LIN {X 0,Y 193.317,Z 565.534,A -85,B 0,C 180,E1 11170.664,E2 11170.664} C_VEL
LIN {X 0,Y 192.779,Z 572.927,A -85,B 0,C 180,E1 11165.955,E2 11165.955} C_VEL
LIN {X 0,Y 192.758,Z 579.081,A -85,B 0,C 180,E1 11160.892,E2 11160.892} C_VEL
LIN {X 0,Y 193.304,Z 583.795,A -85,B 0,C 180,E1 11155.551,E2 11155.551} C_VEL
LIN {X 0,Y 194.84,Z 586.974,A -85,B 0,C 180,E1 11149.952,E2 11149.952} C_VEL
LIN {X 0,Y 197.91,Z 588.494,A -85,B 0,C 180,E1 11144.169,E2 11144.169} C_VEL
LIN {X 0,Y 202.718,Z 588.212,A -85,B 0,C 180,E1 11138.594,E2 11138.594} C_VEL
LIN {X 0,Y 209.71,Z 586.058,A -85,B 0,C 180,E1 11133.068,E2 11133.068} C_VEL
LIN {X 0,Y 218.66,Z 582.103,A -85,B 0,C 180,E1 11127.966,E2 11127.966} C_VEL
LIN {X 0,Y 230.621,Z 575.806,A -85,B 0,C 180,E1 11122.942,E2 11122.942} C_VEL
LIN {X 0,Y 243.425,Z 568.326,A -85,B 0,C 180,E1 11118.835,E2 11118.835} C_VEL
LIN {X 0,Y 227.864,Z 579.481,A -85,B 0,C 180,E1 11114.244,E2 11114.244} C_VEL
LIN {X 0,Y 214.538,Z 589.641,A -85,B 0,C 180,E1 11108.648,E2 11108.648} C_VEL
LIN {X 0,Y 203.983,Z 598.452,A -85,B 0,C 180,E1 11101.966,E2 11101.966} C_VEL
LIN {X 0,Y 197.328,Z 604.793,A -85,B 0,C 180,E1 11095.192,E2 11095.192} C_VEL
LIN {X 0,Y 193.795,Z 608.88,A -85,B 0,C 180,E1 11088.658,E2 11088.658} C_VEL
LIN {X 0,Y 192.5,Z 611.05,A -85,B 0,C 180,E1 11082.298,E2 11082.298} C_VEL
LIN {X 0,Y 192.502,Z 613.904,A -85,B 0,C 180,E1 11076.264,E2 11076.264} C_VEL
LIN {X 0,Y 192.758,Z 614.861,A -85,B 0,C 180,E1 11071.488,E2 11071.488} C_VEL
LIN {X 0,Y 192.704,Z 614.748,A -85,B 0,C 180,E1 11067.325,E2 11067.325} C_VEL
LIN {X 0,Y 192.429,Z 613.273,A -85,B 0,C 180,E1 11062.238,E2 11062.238} C_VEL
LIN {X 0,Y 192.571,Z 610.294,A -85,B 0,C 180,E1 11056.796,E2 11056.796} C_VEL
LIN {X 0,Y 193.943,Z 605.17,A -85,B 0,C 180,E1 11050.737,E2 11050.737} C_VEL
LIN {X 0,Y 196.931,Z 598.058,A -85,B 0,C 180,E1 11044.757,E2 11044.757} C_VEL
LIN {X 0,Y 201.524,Z 589.121,A -85,B 0,C 180,E1 11039.129,E2 11039.129} C_VEL
LIN {X 0,Y 207.508,Z 578.491,A -85,B 0,C 180,E1 11033.998,E2 11033.998} C_VEL
LIN {X 0,Y 214.498,Z 566.341,A -85,B 0,C 180,E1 11029.446,E2 11029.446} C_VEL
LIN {X 0,Y 221.754,Z 553.485,A -85,B 0,C 180,E1 11025.666,E2 11025.666} C_VEL
LIN {X 0,Y 229.612,Z 538.815,A -85,B 0,C 180,E1 11022.248,E2 11022.248} C_VEL
LIN {X 0,Y 237.389,Z 523.208,A -85,B 0,C 180,E1 11019.389,E2 11019.389} C_VEL
LIN {X 0,Y 245.09,Z 506.03,A -85,B 0,C 180,E1 11016.912,E2 11016.912} C_VEL
LIN {X 0,Y 252.259,Z 487.828,A -85,B 0,C 180,E1 11014.871,E2 11014.871} C_VEL
LIN {X 0,Y 258.729,Z 468.548,A -85,B 0,C 180,E1 11013.214,E2 11013.214} C_VEL
LIN {X 0,Y 264.201,Z 448.663,A -85,B 0,C 180,E1 11011.936,E2 11011.936} C_VEL
LIN {X 0,Y 268.521,Z 428.317,A -85,B 0,C 180,E1 11010.995,E2 11010.995} C_VEL
LIN {X 0,Y 271.453,Z 407.696,A -85,B 0,C 180,E1 11010.314,E2 11010.314} C_VEL
LIN {X 0,Y 283.208,Z 264.628,A -85,B 0,C 180,E1 11006.95,E2 11006.95} C_VEL
LIN {X 0,Y 277.161,Z 252.774,A -85,B 0,C 180,E1 11004,E2 11004} C_VEL
LIN {X 0,Y 271.092,Z 241.951,A -85,B 0,C 180,E1 11000.623,E2 11000.623} C_VEL
LIN {X 0,Y 265.539,Z 232.807,A -85,B 0,C 180,E1 10996.966,E2 10996.966} C_VEL
LIN {X 0,Y 261.319,Z 226.484,A -85,B 0,C 180,E1 10993.61,E2 10993.61} C_VEL
LIN {X 0,Y 257.235,Z 220.276,A -85,B 0,C 180,E1 10989.395,E2 10989.395} C_VEL
LIN {X 0,Y 253.535,Z 215.028,A -85,B 0,C 180,E1 10983.391,E2 10983.391} C_VEL
LIN {X 0,Y 252.165,Z 214.003,A -85,B 0,C 180,E1 10977.669,E2 10977.669} C_VEL
LIN {X 0,Y 253.046,Z 214.835,A -85,B 0,C 180,E1 10972.05,E2 10972.05} C_VEL
LIN {X 0,Y 254.504,Z 217.513,A -85,B 0,C 180,E1 10968.671,E2 10968.671} C_VEL
LIN {X 0,Y 256.508,Z 220.315,A -85,B 0,C 180,E1 10965.669,E2 10965.669} C_VEL
LIN {X 0,Y 259.292,Z 224.531,A -85,B 0,C 180,E1 10962.495,E2 10962.495} C_VEL
LIN {X 0,Y 262.787,Z 230.079,A -85,B 0,C 180,E1 10959.335,E2 10959.335} C_VEL
LIN {X 0,Y 266.927,Z 236.838,A -85,B 0,C 180,E1 10956.254,E2 10956.254} C_VEL
LIN {X 0,Y 272.11,Z 245.688,A -85,B 0,C 180,E1 10953.012,E2 10953.012} C_VEL
LIN {X 0,Y 277.72,Z 256.39,A -85,B 0,C 180,E1 10949.971,E2 10949.971} C_VEL
LIN {X 0,Y 282.409,Z 266.043,A -85,B 0,C 180,E1 10947.701,E2 10947.701} C_VEL
LIN {X 0,Y 272.234,Z 400.353,A -85,B 0,C 180,E1 10944.734,E2 10944.734} C_VEL
LIN {X 0,Y 269.376,Z 420.282,A -85,B 0,C 180,E1 10944,E2 10944} C_VEL
LIN {X 0,Y 265.439,Z 439.177,A -85,B 0,C 180,E1 10942.991,E2 10942.991} C_VEL
LIN {X 0,Y 260.23,Z 458.141,A -85,B 0,C 180,E1 10941.608,E2 10941.608} C_VEL
LIN {X 0,Y 254.184,Z 475.871,A -85,B 0,C 180,E1 10939.912,E2 10939.912} C_VEL
LIN {X 0,Y 247.521,Z 492.312,A -85,B 0,C 180,E1 10937.889,E2 10937.889} C_VEL
LIN {X 0,Y 240.101,Z 508.124,A -85,B 0,C 180,E1 10935.403,E2 10935.403} C_VEL
LIN {X 0,Y 232.4,Z 522.631,A -85,B 0,C 180,E1 10932.488,E2 10932.488} C_VEL
LIN {X 0,Y 224.788,Z 535.568,A -85,B 0,C 180,E1 10929.167,E2 10929.167} C_VEL
LIN {X 0,Y 217.062,Z 547.691,A -85,B 0,C 180,E1 10925.153,E2 10925.153} C_VEL
LIN {X 0,Y 209.99,Z 558.111,A -85,B 0,C 180,E1 10920.627,E2 10920.627} C_VEL
LIN {X 0,Y 204.161,Z 566.454,A -85,B 0,C 180,E1 10915.838,E2 10915.838} C_VEL
LIN {X 0,Y 199.4,Z 573.283,A -85,B 0,C 180,E1 10910.547,E2 10910.547} C_VEL
LIN {X 0,Y 195.929,Z 578.505,A -85,B 0,C 180,E1 10904.781,E2 10904.781} C_VEL
LIN {X 0,Y 193.917,Z 581.886,A -85,B 0,C 180,E1 10898.896,E2 10898.896} C_VEL
LIN {X 0,Y 193.081,Z 583.551,A -85,B 0,C 180,E1 10892.966,E2 10892.966} C_VEL
LIN {X 0,Y 193.042,Z 583.608,A -85,B 0,C 180,E1 10887.623,E2 10887.623} C_VEL
LIN {X 0,Y 193.706,Z 582.254,A -85,B 0,C 180,E1 10881.987,E2 10881.987} C_VEL
LIN {X 0,Y 195.505,Z 579.177,A -85,B 0,C 180,E1 10876.09,E2 10876.09} C_VEL
LIN {X 0,Y 198.527,Z 574.566,A -85,B 0,C 180,E1 10870.584,E2 10870.584} C_VEL
LIN {X 0,Y 202.969,Z 568.179,A -85,B 0,C 180,E1 10865.244,E2 10865.244} C_VEL
LIN {X 0,Y 208.843,Z 559.822,A -85,B 0,C 180,E1 10860.136,E2 10860.136} C_VEL
LIN {X 0,Y 215.508,Z 550.105,A -85,B 0,C 180,E1 10855.675,E2 10855.675} C_VEL
LIN {X 0,Y 222.772,Z 538.93,A -85,B 0,C 180,E1 10851.727,E2 10851.727} C_VEL
LIN {X 0,Y 230.701,Z 525.764,A -85,B 0,C 180,E1 10848.129,E2 10848.129} C_VEL
LIN {X 0,Y 238.343,Z 511.77,A -85,B 0,C 180,E1 10845.151,E2 10845.151} C_VEL
LIN {X 0,Y 245.8,Z 496.4,A -85,B 0,C 180,E1 10842.584,E2 10842.584} C_VEL
LIN {X 0,Y 249.129,Z 488.6,A -85,B 0,C 180,E1 10841.47,E2 10841.47} C_VEL
LIN {X 0,Y 242.04,Z 492.975,A -85,B 0,C 180,E1 10840.434,E2 10840.434} C_VEL
LIN {X 0,Y 236.444,Z 495.579,A -85,B 0,C 180,E1 10839.37,E2 10839.37} C_VEL
LIN {X 0,Y 230.606,Z 498.731,A -85,B 0,C 180,E1 10838.318,E2 10838.318} C_VEL
LIN {X 0,Y 225.463,Z 500.858,A -85,B 0,C 180,E1 10837.094,E2 10837.094} C_VEL
LIN {X 0,Y 220.189,Z 503.321,A -85,B 0,C 180,E1 10835.859,E2 10835.859} C_VEL
LIN {X 0,Y 217.063,Z 504.339,A -85,B 0,C 180,E1 10834.92,E2 10834.92} C_VEL
LIN {X 0,Y 212.582,Z 506.314,A -85,B 0,C 180,E1 10833.711,E2 10833.711} C_VEL
LIN {X 0,Y 209.666,Z 507.046,A -85,B 0,C 180,E1 10832.608,E2 10832.608} C_VEL
LIN {X 0,Y 206.241,Z 508.614,A -85,B 0,C 180,E1 10831.574,E2 10831.574} C_VEL
LIN {X 0,Y 204.173,Z 508.704,A -85,B 0,C 180,E1 10830.467,E2 10830.467} C_VEL
LIN {X 0,Y 204.02,Z 508.79,A -85,B 0,C 180,E1 10830.318,E2 10830.318} C_VEL
LIN {X 0,Y 202.338,Z 516.493,A -85,B 0,C 180,E1 10828.545,E2 10828.545} C_VEL
LIN {X 0,Y 200.143,Z 522.205,A -85,B 0,C 180,E1 10827.184,E2 10827.184} C_VEL
LIN {X 0,Y 190.942,Z 536.235,A -85,B 0,C 180,E1 10823.343,E2 10823.343} C_VEL
LIN {X 0,Y 189.307,Z 540.529,A -85,B 0,C 180,E1 10821.886,E2 10821.886} C_VEL
LIN {X 0,Y 187.051,Z 552.693,A -85,B 0,C 180,E1 10817.098,E2 10817.098} C_VEL
LIN {X 0,Y 185.592,Z 562.904,A -85,B 0,C 180,E1 10812.129,E2 10812.129} C_VEL
LIN {X 0,Y 184.867,Z 571.086,A -85,B 0,C 180,E1 10807.147,E2 10807.147} C_VEL
LIN {X 0,Y 184.716,Z 577.509,A -85,B 0,C 180,E1 10802.172,E2 10802.172} C_VEL
LIN {X 0,Y 185.051,Z 582.408,A -85,B 0,C 180,E1 10797.213,E2 10797.213} C_VEL
LIN {X 0,Y 186.206,Z 586.319,A -85,B 0,C 180,E1 10791.665,E2 10791.665} C_VEL
LIN {X 0,Y 188.824,Z 588.824,A -85,B 0,C 180,E1 10785.708,E2 10785.708} C_VEL
LIN {X 0,Y 193.351,Z 589.598,A -85,B 0,C 180,E1 10779.729,E2 10779.729} C_VEL
LIN {X 0,Y 200.077,Z 588.566,A -85,B 0,C 180,E1 10773.912,E2 10773.912} C_VEL
LIN {X 0,Y 209.311,Z 585.545,A -85,B 0,C 180,E1 10768.302,E2 10768.302} C_VEL
LIN {X 0,Y 220.679,Z 580.686,A -85,B 0,C 180,E1 10763.269,E2 10763.269} C_VEL
LIN {X 0,Y 233.542,Z 574.361,A -85,B 0,C 180,E1 10758.947,E2 10758.947} C_VEL
LIN {X 0,Y 217.573,Z 584.638,A -85,B 0,C 180,E1 10753.943,E2 10753.943} C_VEL
LIN {X 0,Y 204.543,Z 593.532,A -85,B 0,C 180,E1 10748.021,E2 10748.021} C_VEL
LIN {X 0,Y 194.71,Z 600.824,A -85,B 0,C 180,E1 10741.243,E2 10741.243} C_VEL
LIN {X 0,Y 188.417,Z 606.097,A -85,B 0,C 180,E1 10734.115,E2 10734.115} C_VEL
LIN {X 0,Y 185.325,Z 609.21,A -85,B 0,C 180,E1 10727.263,E2 10727.263} C_VEL
LIN {X 0,Y 184.505,Z 610.629,A -85,B 0,C 180,E1 10722.203,E2 10722.203} C_VEL
LIN {X 0,Y 184.5,Z 613.253,A -85,B 0,C 180,E1 10716.537,E2 10716.537} C_VEL
LIN {X 0,Y 184.78,Z 614.215,A -85,B 0,C 180,E1 10711.552,E2 10711.552} C_VEL
LIN {X 0,Y 184.721,Z 614.101,A -85,B 0,C 180,E1 10707.21,E2 10707.21} C_VEL
LIN {X 0,Y 184.432,Z 612.619,A -85,B 0,C 180,E1 10701.899,E2 10701.899} C_VEL
LIN {X 0,Y 184.64,Z 609.631,A -85,B 0,C 180,E1 10696.218,E2 10696.218} C_VEL
LIN {X 0,Y 186.147,Z 604.643,A -85,B 0,C 180,E1 10690.047,E2 10690.047} C_VEL
LIN {X 0,Y 189.4,Z 597.551,A -85,B 0,C 180,E1 10683.823,E2 10683.823} C_VEL
LIN {X 0,Y 194.334,Z 588.647,A -85,B 0,C 180,E1 10678.001,E2 10678.001} C_VEL
LIN {X 0,Y 200.48,Z 578.404,A -85,B 0,C 180,E1 10672.884,E2 10672.884} C_VEL
LIN {X 0,Y 207.6,Z 566.726,A -85,B 0,C 180,E1 10668.348,E2 10668.348} C_VEL
LIN {X 0,Y 215.404,Z 553.641,A -85,B 0,C 180,E1 10664.373,E2 10664.373} C_VEL
LIN {X 0,Y 223.585,Z 539.113,A -85,B 0,C 180,E1 10660.911,E2 10660.911} C_VEL
LIN {X 0,Y 231.956,Z 523.045,A -85,B 0,C 180,E1 10657.927,E2 10657.927} C_VEL
LIN {X 0,Y 239.936,Z 505.941,A -85,B 0,C 180,E1 10655.447,E2 10655.447} C_VEL
LIN {X 0,Y 247.343,Z 487.824,A -85,B 0,C 180,E1 10653.413,E2 10653.413} C_VEL
LIN {X 0,Y 253.618,Z 469.905,A -85,B 0,C 180,E1 10651.858,E2 10651.858} C_VEL
LIN {X 0,Y 259.266,Z 450.391,A -85,B 0,C 180,E1 10650.578,E2 10650.578} C_VEL
LIN {X 0,Y 263.774,Z 430.446,A -85,B 0,C 180,E1 10649.631,E2 10649.631} C_VEL
LIN {X 0,Y 266.982,Z 409.697,A -85,B 0,C 180,E1 10648.924,E2 10648.924} C_VEL
LIN {X 0,Y 279.001,Z 268.565,A -85,B 0,C 180,E1 10645.619,E2 10645.619} C_VEL
LIN {X 0,Y 273.685,Z 257.914,A -85,B 0,C 180,E1 10642.84,E2 10642.84} C_VEL
LIN {X 0,Y 267.995,Z 247.578,A -85,B 0,C 180,E1 10639.449,E2 10639.449} C_VEL
LIN {X 0,Y 262.955,Z 239.162,A -85,B 0,C 180,E1 10635.888,E2 10635.888} C_VEL
LIN {X 0,Y 259.587,Z 233.83,A -85,B 0,C 180,E1 10633.022,E2 10633.022} C_VEL
LIN {X 0,Y 255.689,Z 227.8,A -85,B 0,C 180,E1 10628.772,E2 10628.772} C_VEL
LIN {X 0,Y 252.451,Z 222.916,A -85,B 0,C 180,E1 10623.178,E2 10623.178} C_VEL
LIN {X 0,Y 251.185,Z 221.942,A -85,B 0,C 180,E1 10617.49,E2 10617.49} C_VEL
LIN {X 0,Y 252.163,Z 222.852,A -85,B 0,C 180,E1 10611.793,E2 10611.793} C_VEL
LIN {X 0,Y 255.207,Z 228.026,A -85,B 0,C 180,E1 10606.057,E2 10606.057} C_VEL
LIN {X 0,Y 257.892,Z 232.295,A -85,B 0,C 180,E1 10602.863,E2 10602.863} C_VEL
LIN {X 0,Y 261.103,Z 237.568,A -85,B 0,C 180,E1 10599.84,E2 10599.84} C_VEL
LIN {X 0,Y 264.901,Z 244.008,A -85,B 0,C 180,E1 10596.887,E2 10596.887} C_VEL
LIN {X 0,Y 269.754,Z 252.61,A -85,B 0,C 180,E1 10593.708,E2 10593.708} C_VEL
LIN {X 0,Y 275.088,Z 263.184,A -85,B 0,C 180,E1 10590.674,E2 10590.674} C_VEL
LIN {X 0,Y 278.229,Z 270.032,A -85,B 0,C 180,E1 10589.05,E2 10589.05} C_VEL
LIN {X 0,Y 267.961,Z 400.656,A -85,B 0,C 180,E1 10586.167,E2 10586.167} C_VEL
LIN {X 0,Y 265.014,Z 420.58,A -85,B 0,C 180,E1 10585.438,E2 10585.438} C_VEL
LIN {X 0,Y 260.912,Z 439.648,A -85,B 0,C 180,E1 10584.424,E2 10584.424} C_VEL
LIN {X 0,Y 255.622,Z 458.346,A -85,B 0,C 180,E1 10583.069,E2 10583.069} C_VEL
LIN {X 0,Y 249.46,Z 475.906,A -85,B 0,C 180,E1 10581.403,E2 10581.403} C_VEL
LIN {X 0,Y 242.349,Z 492.894,A -85,B 0,C 180,E1 10579.317,E2 10579.317} C_VEL
LIN {X 0,Y 234.567,Z 508.87,A -85,B 0,C 180,E1 10576.792,E2 10576.792} C_VEL
LIN {X 0,Y 226.569,Z 523.345,A -85,B 0,C 180,E1 10573.853,E2 10573.853} C_VEL
LIN {X 0,Y 218.64,Z 536.263,A -85,B 0,C 180,E1 10570.492,E2 10570.492} C_VEL
LIN {X 0,Y 210.558,Z 548.365,A -85,B 0,C 180,E1 10566.409,E2 10566.409} C_VEL
LIN {X 0,Y 203.124,Z 558.772,A -85,B 0,C 180,E1 10561.78,E2 10561.78} C_VEL
LIN {X 0,Y 196.966,Z 567.11,A -85,B 0,C 180,E1 10556.856,E2 10556.856} C_VEL
LIN {X 0,Y 191.903,Z 573.936,A -85,B 0,C 180,E1 10551.388,E2 10551.388} C_VEL
LIN {X 0,Y 188.188,Z 579.155,A -85,B 0,C 180,E1 10545.404,E2 10545.404} C_VEL
LIN {X 0,Y 186.019,Z 582.533,A -85,B 0,C 180,E1 10539.277,E2 10539.277} C_VEL
LIN {X 0,Y 185.114,Z 584.197,A -85,B 0,C 180,E1 10533.094,E2 10533.094} C_VEL
LIN {X 0,Y 185.072,Z 584.253,A -85,B 0,C 180,E1 10527.521,E2 10527.521} C_VEL
LIN {X 0,Y 185.793,Z 582.9,A -85,B 0,C 180,E1 10521.643,E2 10521.643} C_VEL
LIN {X 0,Y 187.735,Z 579.825,A -85,B 0,C 180,E1 10515.502,E2 10515.502} C_VEL
LIN {X 0,Y 190.975,Z 575.216,A -85,B 0,C 180,E1 10509.783,E2 10509.783} C_VEL
LIN {X 0,Y 195.703,Z 568.833,A -85,B 0,C 180,E1 10504.259,E2 10504.259} C_VEL
LIN {X 0,Y 201.919,Z 560.482,A -85,B 0,C 180,E1 10499.002,E2 10499.002} C_VEL
LIN {X 0,Y 209.136,Z 550.488,A -85,B 0,C 180,E1 10494.317,E2 10494.317} C_VEL
LIN {X 0,Y 216.539,Z 539.611,A -85,B 0,C 180,E1 10490.414,E2 10490.414} C_VEL
LIN {X 0,Y 224.808,Z 526.464,A -85,B 0,C 180,E1 10486.768,E2 10486.768} C_VEL
LIN {X 0,Y 232.784,Z 512.434,A -85,B 0,C 180,E1 10483.752,E2 10483.752} C_VEL
LIN {X 0,Y 239.327,Z 499.4,A -85,B 0,C 180,E1 10481.483,E2 10481.483} C_VEL
LIN {X 0,Y 234.464,Z 501.682,A -85,B 0,C 180,E1 10480.616,E2 10480.616} C_VEL
LIN {X 0,Y 227.274,Z 505.075,A -85,B 0,C 180,E1 10479.31,E2 10479.31} C_VEL
LIN {X 0,Y 223.374,Z 506.608,A -85,B 0,C 180,E1 10478.432,E2 10478.432} C_VEL
LIN {X 0,Y 217.338,Z 509.219,A -85,B 0,C 180,E1 10477.062,E2 10477.062} C_VEL
LIN {X 0,Y 214.469,Z 510.161,A -85,B 0,C 180,E1 10476.239,E2 10476.239} C_VEL
LIN {X 0,Y 209.522,Z 512.178,A -85,B 0,C 180,E1 10474.936,E2 10474.936} C_VEL
LIN {X 0,Y 206.412,Z 513.017,A -85,B 0,C 180,E1 10473.853,E2 10473.853} C_VEL
LIN {X 0,Y 202.346,Z 514.592,A -85,B 0,C 180,E1 10472.589,E2 10472.589} C_VEL
LIN {X 0,Y 199.929,Z 515.04,A -85,B 0,C 180,E1 10471.508,E2 10471.508} C_VEL
LIN {X 0,Y 196.368,Z 516.493,A -85,B 0,C 180,E1 10470.271,E2 10470.271} C_VEL
LIN {X 0,Y 194.54,Z 516.398,A -85,B 0,C 180,E1 10469.061,E2 10469.061} C_VEL
LIN {X 0,Y 191.211,Z 531.464,A -85,B 0,C 180,E1 10464.895,E2 10464.895} C_VEL
LIN {X 0,Y 189.307,Z 540.529,A -85,B 0,C 180,E1 10461.886,E2 10461.886} C_VEL
LIN {X 0,Y 187.375,Z 545.397,A -85,B 0,C 180,E1 10460.139,E2 10460.139} C_VEL
LIN {X 0,Y 181.034,Z 554.138,A -85,B 0,C 180,E1 10456.597,E2 10456.597} C_VEL
LIN {X 0,Y 178.309,Z 558.788,A -85,B 0,C 180,E1 10454.318,E2 10454.318} C_VEL
LIN {X 0,Y 177.868,Z 560.491,A -85,B 0,C 180,E1 10453.401,E2 10453.401} C_VEL
LIN {X 0,Y 176.963,Z 569.384,A -85,B 0,C 180,E1 10448.121,E2 10448.121} C_VEL
LIN {X 0,Y 176.712,Z 576.37,A -85,B 0,C 180,E1 10442.92,E2 10442.92} C_VEL
LIN {X 0,Y 177.023,Z 582.064,A -85,B 0,C 180,E1 10437.411,E2 10437.411} C_VEL
LIN {X 0,Y 178.188,Z 586.399,A -85,B 0,C 180,E1 10431.612,E2 10431.612} C_VEL
LIN {X 0,Y 180.965,Z 589.377,A -85,B 0,C 180,E1 10425.277,E2 10425.277} C_VEL
LIN {X 0,Y 185.62,Z 590.598,A -85,B 0,C 180,E1 10419.176,E2 10419.176} C_VEL
LIN {X 0,Y 192.643,Z 590.095,A -85,B 0,C 180,E1 10413.158,E2 10413.158} C_VEL
LIN {X 0,Y 202.279,Z 587.738,A -85,B 0,C 180,E1 10407.4,E2 10407.4} C_VEL
LIN {X 0,Y 214.1,Z 583.619,A -85,B 0,C 180,E1 10402.282,E2 10402.282} C_VEL
LIN {X 0,Y 223.555,Z 579.723,A -85,B 0,C 180,E1 10399.054,E2 10399.054} C_VEL
LIN {X 0,Y 206.701,Z 589.398,A -85,B 0,C 180,E1 10393.386,E2 10393.386} C_VEL
LIN {X 0,Y 193.671,Z 597.299,A -85,B 0,C 180,E1 10386.791,E2 10386.791} C_VEL
LIN {X 0,Y 184.545,Z 603.289,A -85,B 0,C 180,E1 10379.542,E2 10379.542} C_VEL
LIN {X 0,Y 179.137,Z 607.238,A -85,B 0,C 180,E1 10372.101,E2 10372.101} C_VEL
LIN {X 0,Y 176.86,Z 609.138,A -85,B 0,C 180,E1 10365.075,E2 10365.075} C_VEL
LIN {X 0,Y 176.505,Z 610.321,A -85,B 0,C 180,E1 10362.101,E2 10362.101} C_VEL
LIN {X 0,Y 176.543,Z 612.763,A -85,B 0,C 180,E1 10356.179,E2 10356.179} C_VEL
LIN {X 0,Y 176.814,Z 613.596,A -85,B 0,C 180,E1 10351.298,E2 10351.298} C_VEL
LIN {X 0,Y 176.717,Z 613.425,A -85,B 0,C 180,E1 10346.759,E2 10346.759} C_VEL
LIN {X 0,Y 176.43,Z 611.835,A -85,B 0,C 180,E1 10341.201,E2 10341.201} C_VEL
LIN {X 0,Y 176.824,Z 608.512,A -85,B 0,C 180,E1 10334.926,E2 10334.926} C_VEL
LIN {X 0,Y 178.632,Z 603.499,A -85,B 0,C 180,E1 10328.667,E2 10328.667} C_VEL
LIN {X 0,Y 182.117,Z 596.705,A -85,B 0,C 180,E1 10322.539,E2 10322.539} C_VEL
LIN {X 0,Y 187.363,Z 587.965,A -85,B 0,C 180,E1 10316.659,E2 10316.659} C_VEL
LIN {X 0,Y 193.938,Z 577.713,A -85,B 0,C 180,E1 10311.407,E2 10311.407} C_VEL
LIN {X 0,Y 201.498,Z 566.022,A -85,B 0,C 180,E1 10306.785,E2 10306.785} C_VEL
LIN {X 0,Y 209.711,Z 552.917,A -85,B 0,C 180,E1 10302.76,E2 10302.76} C_VEL
LIN {X 0,Y 218.286,Z 538.364,A -85,B 0,C 180,E1 10299.279,E2 10299.279} C_VEL
LIN {X 0,Y 227.004,Z 522.259,A -85,B 0,C 180,E1 10296.293,E2 10296.293} C_VEL
LIN {X 0,Y 235.257,Z 505.164,A -85,B 0,C 180,E1 10293.831,E2 10293.831} C_VEL
LIN {X 0,Y 242.948,Z 486.902,A -85,B 0,C 180,E1 10291.807,E2 10291.807} C_VEL
LIN {X 0,Y 249.828,Z 467.605,A -85,B 0,C 180,E1 10290.181,E2 10290.181} C_VEL
LIN {X 0,Y 255.619,Z 447.664,A -85,B 0,C 180,E1 10288.935,E2 10288.935} C_VEL
LIN {X 0,Y 260.164,Z 427.176,A -85,B 0,C 180,E1 10288.016,E2 10288.016} C_VEL
LIN {X 0,Y 263.229,Z 406.407,A -85,B 0,C 180,E1 10287.35,E2 10287.35} C_VEL
LIN {X 0,Y 274.88,Z 272.405,A -85,B 0,C 180,E1 10284.212,E2 10284.212} C_VEL
LIN {X 0,Y 269.725,Z 262.026,A -85,B 0,C 180,E1 10281.301,E2 10281.301} C_VEL
LIN {X 0,Y 265.379,Z 253.923,A -85,B 0,C 180,E1 10278.507,E2 10278.507} C_VEL
LIN {X 0,Y 260.795,Z 245.992,A -85,B 0,C 180,E1 10275.055,E2 10275.055} C_VEL
LIN {X 0,Y 257.248,Z 240.052,A -85,B 0,C 180,E1 10271.774,E2 10271.774} C_VEL
LIN {X 0,Y 254.343,Z 235.501,A -85,B 0,C 180,E1 10268.363,E2 10268.363} C_VEL
LIN {X 0,Y 251.37,Z 230.804,A -85,B 0,C 180,E1 10262.964,E2 10262.964} C_VEL
LIN {X 0,Y 250.206,Z 229.881,A -85,B 0,C 180,E1 10257.443,E2 10257.443} C_VEL
LIN {X 0,Y 251.111,Z 230.75,A -85,B 0,C 180,E1 10251.989,E2 10251.989} C_VEL
LIN {X 0,Y 253.908,Z 235.735,A -85,B 0,C 180,E1 10246.449,E2 10246.449} C_VEL
LIN {X 0,Y 256.4,Z 239.863,A -85,B 0,C 180,E1 10243.344,E2 10243.344} C_VEL
LIN {X 0,Y 259.566,Z 245.269,A -85,B 0,C 180,E1 10240.243,E2 10240.243} C_VEL
LIN {X 0,Y 262.966,Z 251.287,A -85,B 0,C 180,E1 10237.486,E2 10237.486} C_VEL
LIN {X 0,Y 267.591,Z 259.871,A -85,B 0,C 180,E1 10234.314,E2 10234.314} C_VEL
LIN {X 0,Y 272.681,Z 270.347,A -85,B 0,C 180,E1 10231.291,E2 10231.291} C_VEL
LIN {X 0,Y 274.215,Z 273.918,A -85,B 0,C 180,E1 10230.441,E2 10230.441} C_VEL
LIN {X 0,Y 263.859,Z 400.959,A -85,B 0,C 180,E1 10227.646,E2 10227.646} C_VEL
LIN {X 0,Y 260.824,Z 420.877,A -85,B 0,C 180,E1 10226.923,E2 10226.923} C_VEL
LIN {X 0,Y 256.555,Z 440.118,A -85,B 0,C 180,E1 10225.908,E2 10225.908} C_VEL
LIN {X 0,Y 251.018,Z 459.041,A -85,B 0,C 180,E1 10224.542,E2 10224.542} C_VEL
LIN {X 0,Y 244.576,Z 476.766,A -85,B 0,C 180,E1 10222.859,E2 10222.859} C_VEL
LIN {X 0,Y 237.33,Z 493.48,A -85,B 0,C 180,E1 10220.806,E2 10220.806} C_VEL
LIN {X 0,Y 229.177,Z 509.608,A -85,B 0,C 180,E1 10218.246,E2 10218.246} C_VEL
LIN {X 0,Y 220.874,Z 524.055,A -85,B 0,C 180,E1 10215.29,E2 10215.29} C_VEL
LIN {X 0,Y 212.616,Z 536.957,A -85,B 0,C 180,E1 10211.893,E2 10211.893} C_VEL
LIN {X 0,Y 204.16,Z 549.037,A -85,B 0,C 180,E1 10207.745,E2 10207.745} C_VEL
LIN {X 0,Y 196.347,Z 559.432,A -85,B 0,C 180,E1 10203.014,E2 10203.014} C_VEL
LIN {X 0,Y 189.836,Z 567.766,A -85,B 0,C 180,E1 10197.951,E2 10197.951} C_VEL
LIN {X 0,Y 184.452,Z 574.589,A -85,B 0,C 180,E1 10192.297,E2 10192.297} C_VEL
LIN {X 0,Y 180.472,Z 579.804,A -85,B 0,C 180,E1 10186.08,E2 10186.08} C_VEL
LIN {X 0,Y 178.13,Z 583.181,A -85,B 0,C 180,E1 10179.692,E2 10179.692} C_VEL
LIN {X 0,Y 177.148,Z 584.842,A -85,B 0,C 180,E1 10173.234,E2 10173.234} C_VEL
LIN {X 0,Y 177.103,Z 584.898,A -85,B 0,C 180,E1 10167.409,E2 10167.409} C_VEL
LIN {X 0,Y 177.887,Z 583.547,A -85,B 0,C 180,E1 10161.269,E2 10161.269} C_VEL
LIN {X 0,Y 179.984,Z 580.474,A -85,B 0,C 180,E1 10154.863,E2 10154.863} C_VEL
LIN {X 0,Y 183.463,Z 575.868,A -85,B 0,C 180,E1 10148.917,E2 10148.917} C_VEL
LIN {X 0,Y 188.501,Z 569.488,A -85,B 0,C 180,E1 10143.199,E2 10143.199} C_VEL
LIN {X 0,Y 195.081,Z 561.141,A -85,B 0,C 180,E1 10137.787,E2 10137.787} C_VEL
LIN {X 0,Y 202.674,Z 551.154,A -85,B 0,C 180,E1 10132.994,E2 10132.994} C_VEL
LIN {X 0,Y 210.427,Z 540.29,A -85,B 0,C 180,E1 10129.024,E2 10129.024} C_VEL
LIN {X 0,Y 219.049,Z 527.164,A -85,B 0,C 180,E1 10125.335,E2 10125.335} C_VEL
LIN {X 0,Y 227.377,Z 513.088,A -85,B 0,C 180,E1 10122.284,E2 10122.284} C_VEL
LIN {X 0,Y 229.56,Z 508.927,A -85,B 0,C 180,E1 10121.457,E2 10121.457} C_VEL
LIN {X 0,Y 219.833,Z 512.854,A -85,B 0,C 180,E1 10119.551,E2 10119.551} C_VEL
LIN {X 0,Y 213.026,Z 515.339,A -85,B 0,C 180,E1 10117.943,E2 10117.943} C_VEL
LIN {X 0,Y 205.719,Z 518.037,A -85,B 0,C 180,E1 10116.023,E2 10116.023} C_VEL
LIN {X 0,Y 202.395,Z 519.055,A -85,B 0,C 180,E1 10114.964,E2 10114.964} C_VEL
LIN {X 0,Y 197.763,Z 520.538,A -85,B 0,C 180,E1 10113.442,E2 10113.442} C_VEL
LIN {X 0,Y 196.044,Z 520.903,A -85,B 0,C 180,E1 10112.727,E2 10112.727} C_VEL
LIN {X 0,Y 192.183,Z 522.245,A -85,B 0,C 180,E1 10111.351,E2 10111.351} C_VEL
LIN {X 0,Y 189.586,Z 522.741,A -85,B 0,C 180,E1 10110.068,E2 10110.068} C_VEL
LIN {X 0,Y 186.619,Z 523.776,A -85,B 0,C 180,E1 10108.83,E2 10108.83} C_VEL
LIN {X 0,Y 185.02,Z 523.761,A -85,B 0,C 180,E1 10107.565,E2 10107.565} C_VEL
LIN {X 0,Y 182.015,Z 537.326,A -85,B 0,C 180,E1 10103.299,E2 10103.299} C_VEL
LIN {X 0,Y 179.555,Z 549.787,A -85,B 0,C 180,E1 10098.507,E2 10098.507} C_VEL
LIN {X 0,Y 177.868,Z 560.491,A -85,B 0,C 180,E1 10093.401,E2 10093.401} C_VEL
LIN {X 0,Y 176.418,Z 564.353,A -85,B 0,C 180,E1 10091.256,E2 10091.256} C_VEL
LIN {X 0,Y 171.813,Z 570.066,A -85,B 0,C 180,E1 10087.549,E2 10087.549} C_VEL
LIN {X 0,Y 169.089,Z 573.977,A -85,B 0,C 180,E1 10084.554,E2 10084.554} C_VEL
LIN {X 0,Y 168.72,Z 575.677,A -85,B 0,C 180,E1 10083.161,E2 10083.161} C_VEL
LIN {X 0,Y 168.998,Z 581.492,A -85,B 0,C 180,E1 10077.627,E2 10077.627} C_VEL
LIN {X 0,Y 170.167,Z 586.255,A -85,B 0,C 180,E1 10071.554,E2 10071.554} C_VEL
LIN {X 0,Y 173.037,Z 589.741,A -85,B 0,C 180,E1 10064.929,E2 10064.929} C_VEL
LIN {X 0,Y 178.192,Z 591.527,A -85,B 0,C 180,E1 10058.265,E2 10058.265} C_VEL
LIN {X 0,Y 186.053,Z 591.488,A -85,B 0,C 180,E1 10051.777,E2 10051.777} C_VEL
LIN {X 0,Y 196.305,Z 589.582,A -85,B 0,C 180,E1 10045.926,E2 10045.926} C_VEL
LIN {X 0,Y 209.374,Z 585.763,A -85,B 0,C 180,E1 10040.571,E2 10040.571} C_VEL
LIN {X 0,Y 213.47,Z 584.423,A -85,B 0,C 180,E1 10039.154,E2 10039.154} C_VEL
LIN {X 0,Y 197.523,Z 592.473,A -85,B 0,C 180,E1 10033.508,E2 10033.508} C_VEL
LIN {X 0,Y 184.57,Z 599.306,A -85,B 0,C 180,E1 10026.579,E2 10026.579} C_VEL
LIN {X 0,Y 175.651,Z 604.294,A -85,B 0,C 180,E1 10018.939,E2 10018.939} C_VEL
LIN {X 0,Y 170.68,Z 607.256,A -85,B 0,C 180,E1 10011.299,E2 10011.299} C_VEL
LIN {X 0,Y 168.827,Z 608.57,A -85,B 0,C 180,E1 10004.756,E2 10004.756} C_VEL
LIN {X 0,Y 168.456,Z 611.588,A -85,B 0,C 180,E1 9998.192,E2 9998.192} C_VEL
LIN {X 0,Y 168.772,Z 612.84,A -85,B 0,C 180,E1 9992.719,E2 9992.719} C_VEL
LIN {X 0,Y 168.822,Z 612.92,A -85,B 0,C 180,E1 9988.305,E2 9988.305} C_VEL
LIN {X 0,Y 168.52,Z 612.019,A -85,B 0,C 180,E1 9983.187,E2 9983.187} C_VEL
LIN {X 0,Y 168.567,Z 609.452,A -85,B 0,C 180,E1 9976.976,E2 9976.976} C_VEL
LIN {X 0,Y 170.039,Z 604.856,A -85,B 0,C 180,E1 9970.062,E2 9970.062} C_VEL
LIN {X 0,Y 173.413,Z 598.324,A -85,B 0,C 180,E1 9963.276,E2 9963.276} C_VEL
LIN {X 0,Y 178.508,Z 590.213,A -85,B 0,C 180,E1 9957.093,E2 9957.093} C_VEL
LIN {X 0,Y 185.022,Z 580.649,A -85,B 0,C 180,E1 9951.58,E2 9951.58} C_VEL
LIN {X 0,Y 192.576,Z 569.714,A -85,B 0,C 180,E1 9946.74,E2 9946.74} C_VEL
LIN {X 0,Y 201.397,Z 556.587,A -85,B 0,C 180,E1 9942.295,E2 9942.295} C_VEL
LIN {X 0,Y 210.699,Z 541.805,A -85,B 0,C 180,E1 9938.467,E2 9938.467} C_VEL
LIN {X 0,Y 219.599,Z 526.462,A -85,B 0,C 180,E1 9935.415,E2 9935.415} C_VEL
LIN {X 0,Y 228.391,Z 509.495,A -85,B 0,C 180,E1 9932.806,E2 9932.806} C_VEL
LIN {X 0,Y 236.567,Z 491.433,A -85,B 0,C 180,E1 9930.676,E2 9930.676} C_VEL
LIN {X 0,Y 243.996,Z 472.124,A -85,B 0,C 180,E1 9928.947,E2 9928.947} C_VEL
LIN {X 0,Y 250.245,Z 452.3,A -85,B 0,C 180,E1 9927.628,E2 9927.628} C_VEL
LIN {X 0,Y 255.331,Z 431.55,A -85,B 0,C 180,E1 9926.64,E2 9926.64} C_VEL
LIN {X 0,Y 258.902,Z 410.261,A -85,B 0,C 180,E1 9925.916,E2 9925.916} C_VEL
LIN {X 0,Y 270.969,Z 276.497,A -85,B 0,C 180,E1 9922.795,E2 9922.795} C_VEL
LIN {X 0,Y 266.119,Z 266.536,A -85,B 0,C 180,E1 9919.821,E2 9919.821} C_VEL
LIN {X 0,Y 261.794,Z 258.279,A -85,B 0,C 180,E1 9916.759,E2 9916.759} C_VEL
LIN {X 0,Y 257.534,Z 250.657,A -85,B 0,C 180,E1 9913.127,E2 9913.127} C_VEL
LIN {X 0,Y 254.614,Z 246.026,A -85,B 0,C 180,E1 9910.064,E2 9910.064} C_VEL
LIN {X 0,Y 253.011,Z 243.202,A -85,B 0,C 180,E1 9907.95,E2 9907.95} C_VEL
LIN {X 0,Y 250.293,Z 238.692,A -85,B 0,C 180,E1 9902.747,E2 9902.747} C_VEL
LIN {X 0,Y 249.219,Z 237.818,A -85,B 0,C 180,E1 9897.24,E2 9897.24} C_VEL
LIN {X 0,Y 250.061,Z 238.648,A -85,B 0,C 180,E1 9892.186,E2 9892.186} C_VEL
LIN {X 0,Y 252.699,Z 243.591,A -85,B 0,C 180,E1 9886.732,E2 9886.732} C_VEL
LIN {X 0,Y 255.026,Z 247.618,A -85,B 0,C 180,E1 9883.72,E2 9883.72} C_VEL
LIN {X 0,Y 257.863,Z 252.649,A -85,B 0,C 180,E1 9880.815,E2 9880.815} C_VEL
LIN {X 0,Y 261.153,Z 258.74,A -85,B 0,C 180,E1 9878.022,E2 9878.022} C_VEL
LIN {X 0,Y 265.61,Z 267.447,A -85,B 0,C 180,E1 9874.825,E2 9874.825} C_VEL
LIN {X 0,Y 270.376,Z 277.648,A -85,B 0,C 180,E1 9871.878,E2 9871.878} C_VEL
LIN {X 0,Y 259.94,Z 401.262,A -85,B 0,C 180,E1 9869.171,E2 9869.171} C_VEL
LIN {X 0,Y 256.792,Z 421.283,A -85,B 0,C 180,E1 9868.451,E2 9868.451} C_VEL
LIN {X 0,Y 252.556,Z 439.917,A -85,B 0,C 180,E1 9867.483,E2 9867.483} C_VEL
LIN {X 0,Y 246.851,Z 458.985,A -85,B 0,C 180,E1 9866.131,E2 9866.131} C_VEL
LIN {X 0,Y 240.203,Z 476.8,A -85,B 0,C 180,E1 9864.464,E2 9864.464} C_VEL
LIN {X 0,Y 232.483,Z 494.055,A -85,B 0,C 180,E1 9862.358,E2 9862.358} C_VEL
LIN {X 0,Y 224.261,Z 509.795,A -85,B 0,C 180,E1 9859.871,E2 9859.871} C_VEL
LIN {X 0,Y 215.324,Z 524.759,A -85,B 0,C 180,E1 9856.802,E2 9856.802} C_VEL
LIN {X 0,Y 206.726,Z 537.646,A -85,B 0,C 180,E1 9853.375,E2 9853.375} C_VEL
LIN {X 0,Y 197.88,Z 549.707,A -85,B 0,C 180,E1 9849.166,E2 9849.166} C_VEL
LIN {X 0,Y 190.093,Z 559.59,A -85,B 0,C 180,E1 9844.613,E2 9844.613} C_VEL
LIN {X 0,Y 182.781,Z 568.422,A -85,B 0,C 180,E1 9839.131,E2 9839.131} C_VEL
LIN {X 0,Y 177.052,Z 575.241,A -85,B 0,C 180,E1 9833.283,E2 9833.283} C_VEL
LIN {X 0,Y 172.782,Z 580.453,A -85,B 0,C 180,E1 9826.816,E2 9826.816} C_VEL
LIN {X 0,Y 170.251,Z 583.828,A -85,B 0,C 180,E1 9820.145,E2 9820.145} C_VEL
LIN {X 0,Y 169.183,Z 585.488,A -85,B 0,C 180,E1 9813.386,E2 9813.386} C_VEL
LIN {X 0,Y 169.135,Z 585.543,A -85,B 0,C 180,E1 9807.287,E2 9807.287} C_VEL
LIN {X 0,Y 169.988,Z 584.193,A -85,B 0,C 180,E1 9800.86,E2 9800.86} C_VEL
LIN {X 0,Y 172.258,Z 581.122,A -85,B 0,C 180,E1 9794.166,E2 9794.166} C_VEL
LIN {X 0,Y 176.238,Z 576.23,A -85,B 0,C 180,E1 9787.657,E2 9787.657} C_VEL
LIN {X 0,Y 181.696,Z 569.754,A -85,B 0,C 180,E1 9781.752,E2 9781.752} C_VEL
LIN {X 0,Y 188.44,Z 561.674,A -85,B 0,C 180,E1 9776.414,E2 9776.414} C_VEL
LIN {X 0,Y 196.328,Z 551.821,A -85,B 0,C 180,E1 9771.585,E2 9771.585} C_VEL
LIN {X 0,Y 204.983,Z 540.224,A -85,B 0,C 180,E1 9767.31,E2 9767.31} C_VEL
LIN {X 0,Y 213.435,Z 527.865,A -85,B 0,C 180,E1 9763.825,E2 9763.825} C_VEL
LIN {X 0,Y 219.988,Z 517.27,A -85,B 0,C 180,E1 9761.39,E2 9761.39} C_VEL
LIN {X 0,Y 212.229,Z 520.235,A -85,B 0,C 180,E1 9759.847,E2 9759.847} C_VEL
LIN {X 0,Y 207.67,Z 521.759,A -85,B 0,C 180,E1 9758.749,E2 9758.749} C_VEL
LIN {X 0,Y 201.149,Z 523.836,A -85,B 0,C 180,E1 9756.975,E2 9756.975} C_VEL
LIN {X 0,Y 193.657,Z 526.132,A -85,B 0,C 180,E1 9754.607,E2 9754.607} C_VEL
LIN {X 0,Y 191.025,Z 526.904,A -85,B 0,C 180,E1 9753.668,E2 9753.668} C_VEL
LIN {X 0,Y 186.823,Z 528.017,A -85,B 0,C 180,E1 9751.995,E2 9751.995} C_VEL
LIN {X 0,Y 185.126,Z 528.414,A -85,B 0,C 180,E1 9751.232,E2 9751.232} C_VEL
LIN {X 0,Y 181.649,Z 529.402,A -85,B 0,C 180,E1 9749.696,E2 9749.696} C_VEL
LIN {X 0,Y 179.745,Z 529.705,A -85,B 0,C 180,E1 9748.581,E2 9748.581} C_VEL
LIN {X 0,Y 176.982,Z 530.583,A -85,B 0,C 180,E1 9747.234,E2 9747.234} C_VEL
LIN {X 0,Y 175.571,Z 530.503,A -85,B 0,C 180,E1 9745.919,E2 9745.919} C_VEL
LIN {X 0,Y 172.65,Z 544.03,A -85,B 0,C 180,E1 9741.043,E2 9741.043} C_VEL
LIN {X 0,Y 170.574,Z 555.433,A -85,B 0,C 180,E1 9735.981,E2 9735.981} C_VEL
LIN {X 0,Y 169.284,Z 565.331,A -85,B 0,C 180,E1 9730.551,E2 9730.551} C_VEL
LIN {X 0,Y 168.754,Z 573.291,A -85,B 0,C 180,E1 9725.1,E2 9725.1} C_VEL
LIN {X 0,Y 168.72,Z 575.677,A -85,B 0,C 180,E1 9723.161,E2 9723.161} C_VEL
LIN {X 0,Y 167.998,Z 578.101,A -85,B 0,C 180,E1 9721.068,E2 9721.068} C_VEL
LIN {X 0,Y 164.994,Z 581.482,A -85,B 0,C 180,E1 9717.549,E2 9717.549} C_VEL
LIN {X 0,Y 162.125,Z 584.773,A -85,B 0,C 180,E1 9713.273,E2 9713.273} C_VEL
LIN {X 0,Y 162.13,Z 586.006,A -85,B 0,C 180,E1 9711.543,E2 9711.543} C_VEL
LIN {X 0,Y 165.11,Z 589.987,A -85,B 0,C 180,E1 9704.548,E2 9704.548} C_VEL
LIN {X 0,Y 170.487,Z 592.272,A -85,B 0,C 180,E1 9697.592,E2 9697.592} C_VEL
LIN {X 0,Y 178.259,Z 592.802,A -85,B 0,C 180,E1 9691.16,E2 9691.16} C_VEL
LIN {X 0,Y 188.83,Z 591.615,A -85,B 0,C 180,E1 9685.121,E2 9685.121} C_VEL
LIN {X 0,Y 202.281,Z 588.608,A -85,B 0,C 180,E1 9679.646,E2 9679.646} C_VEL
LIN {X 0,Y 203.259,Z 588.377,A -85,B 0,C 180,E1 9679.251,E2 9679.251} C_VEL
LIN {X 0,Y 187.764,Z 595.27,A -85,B 0,C 180,E1 9673.39,E2 9673.39} C_VEL
LIN {X 0,Y 174.629,Z 601.221,A -85,B 0,C 180,E1 9665.736,E2 9665.736} C_VEL
LIN {X 0,Y 165.992,Z 605.237,A -85,B 0,C 180,E1 9657.247,E2 9657.247} C_VEL
LIN {X 0,Y 161.722,Z 607.136,A -85,B 0,C 180,E1 9648.756,E2 9648.756} C_VEL
LIN {X 0,Y 161.107,Z 607.482,A -85,B 0,C 180,E1 9646.219,E2 9646.219} C_VEL
LIN {X 0,Y 160.448,Z 610.675,A -85,B 0,C 180,E1 9639.327,E2 9639.327} C_VEL
LIN {X 0,Y 160.739,Z 612.134,A -85,B 0,C 180,E1 9633.569,E2 9633.569} C_VEL
LIN {X 0,Y 160.871,Z 612.327,A -85,B 0,C 180,E1 9628.934,E2 9628.934} C_VEL
LIN {X 0,Y 160.585,Z 611.61,A -85,B 0,C 180,E1 9623.926,E2 9623.926} C_VEL
LIN {X 0,Y 160.539,Z 609.33,A -85,B 0,C 180,E1 9617.412,E2 9617.412} C_VEL
LIN {X 0,Y 161.838,Z 605.302,A -85,B 0,C 180,E1 9610.514,E2 9610.514} C_VEL
LIN {X 0,Y 165.152,Z 599.172,A -85,B 0,C 180,E1 9603.387,E2 9603.387} C_VEL
LIN {X 0,Y 170.614,Z 590.994,A -85,B 0,C 180,E1 9596.576,E2 9596.576} C_VEL
LIN {X 0,Y 177.753,Z 581.162,A -85,B 0,C 180,E1 9590.537,E2 9590.537} C_VEL
LIN {X 0,Y 186.129,Z 569.731,A -85,B 0,C 180,E1 9585.277,E2 9585.277} C_VEL
LIN {X 0,Y 195.357,Z 556.722,A -85,B 0,C 180,E1 9580.761,E2 9580.761} C_VEL
LIN {X 0,Y 205.043,Z 542.083,A -85,B 0,C 180,E1 9576.9,E2 9576.9} C_VEL
LIN {X 0,Y 214.606,Z 526.28,A -85,B 0,C 180,E1 9573.736,E2 9573.736} C_VEL
LIN {X 0,Y 223.703,Z 509.376,A -85,B 0,C 180,E1 9571.142,E2 9571.142} C_VEL
LIN {X 0,Y 232.136,Z 491.388,A -85,B 0,C 180,E1 9569.034,E2 9569.034} C_VEL
LIN {X 0,Y 239.353,Z 473.295,A -85,B 0,C 180,E1 9567.42,E2 9567.42} C_VEL
LIN {X 0,Y 245.596,Z 454.411,A -85,B 0,C 180,E1 9566.148,E2 9566.148} C_VEL
LIN {X 0,Y 250.757,Z 434.669,A -85,B 0,C 180,E1 9565.18,E2 9565.18} C_VEL
LIN {X 0,Y 254.58,Z 414.169,A -85,B 0,C 180,E1 9564.455,E2 9564.455} C_VEL
LIN {X 0,Y 257.639,Z 385.719,A -85,B 0,C 180,E1 9563.742,E2 9563.742} C_VEL
LIN {X 0,Y 267.225,Z 280.615,A -85,B 0,C 180,E1 9561.338,E2 9561.338} C_VEL
LIN {X 0,Y 262.048,Z 269.762,A -85,B 0,C 180,E1 9557.83,E2 9557.83} C_VEL
LIN {X 0,Y 257.648,Z 261.379,A -85,B 0,C 180,E1 9554.266,E2 9554.266} C_VEL
LIN {X 0,Y 254.179,Z 255.118,A -85,B 0,C 180,E1 9550.769,E2 9550.769} C_VEL
LIN {X 0,Y 251.695,Z 250.901,A -85,B 0,C 180,E1 9547.532,E2 9547.532} C_VEL
LIN {X 0,Y 249.228,Z 246.58,A -85,B 0,C 180,E1 9542.529,E2 9542.529} C_VEL
LIN {X 0,Y 248.243,Z 245.754,A -85,B 0,C 180,E1 9536.998,E2 9536.998} C_VEL
LIN {X 0,Y 249.083,Z 246.732,A -85,B 0,C 180,E1 9532.155,E2 9532.155} C_VEL
LIN {X 0,Y 251.433,Z 251.299,A -85,B 0,C 180,E1 9527.132,E2 9527.132} C_VEL
LIN {X 0,Y 253.573,Z 255.185,A -85,B 0,C 180,E1 9524.212,E2 9524.212} C_VEL
LIN {X 0,Y 256.467,Z 260.549,A -85,B 0,C 180,E1 9521.12,E2 9521.12} C_VEL
LIN {X 0,Y 259.545,Z 266.549,A -85,B 0,C 180,E1 9518.413,E2 9518.413} C_VEL
LIN {X 0,Y 263.653,Z 275.005,A -85,B 0,C 180,E1 9515.344,E2 9515.344} C_VEL
LIN {X 0,Y 266.675,Z 281.913,A -85,B 0,C 180,E1 9513.341,E2 9513.341} C_VEL
LIN {X 0,Y 256.186,Z 401.724,A -85,B 0,C 180,E1 9510.736,E2 9510.736} C_VEL
LIN {X 0,Y 252.948,Z 421.686,A -85,B 0,C 180,E1 9510.026,E2 9510.026} C_VEL
LIN {X 0,Y 248.383,Z 441.052,A -85,B 0,C 180,E1 9509.025,E2 9509.025} C_VEL
LIN {X 0,Y 242.513,Z 459.939,A -85,B 0,C 180,E1 9507.689,E2 9507.689} C_VEL
LIN {X 0,Y 235.669,Z 477.659,A -85,B 0,C 180,E1 9506.038,E2 9506.038} C_VEL
LIN {X 0,Y 227.808,Z 494.638,A -85,B 0,C 180,E1 9503.975,E2 9503.975} C_VEL
LIN {X 0,Y 219.203,Z 510.534,A -85,B 0,C 180,E1 9501.466,E2 9501.466} C_VEL
LIN {X 0,Y 210.553,Z 524.534,A -85,B 0,C 180,E1 9498.613,E2 9498.613} C_VEL
LIN {X 0,Y 201.555,Z 537.532,A -85,B 0,C 180,E1 9495.182,E2 9495.182} C_VEL
LIN {X 0,Y 192.763,Z 549.063,A -85,B 0,C 180,E1 9491.201,E2 9491.201} C_VEL
LIN {X 0,Y 184.443,Z 559.157,A -85,B 0,C 180,E1 9486.603,E2 9486.603} C_VEL
LIN {X 0,Y 176.92,Z 567.789,A -85,B 0,C 180,E1 9481.325,E2 9481.325} C_VEL
LIN {X 0,Y 170.85,Z 574.567,A -85,B 0,C 180,E1 9475.66,E2 9475.66} C_VEL
LIN {X 0,Y 166.087,Z 579.933,A -85,B 0,C 180,E1 9469.333,E2 9469.333} C_VEL
LIN {X 0,Y 162.903,Z 583.75,A -85,B 0,C 180,E1 9462.403,E2 9462.403} C_VEL
LIN {X 0,Y 161.379,Z 585.825,A -85,B 0,C 180,E1 9455.33,E2 9455.33} C_VEL
LIN {X 0,Y 161.108,Z 586.27,A -85,B 0,C 180,E1 9448.575,E2 9448.575} C_VEL
LIN {X 0,Y 161.8,Z 585.259,A -85,B 0,C 180,E1 9441.827,E2 9441.827} C_VEL
LIN {X 0,Y 163.788,Z 582.737,A -85,B 0,C 180,E1 9435.142,E2 9435.142} C_VEL
LIN {X 0,Y 167.595,Z 578.316,A -85,B 0,C 180,E1 9428.289,E2 9428.289} C_VEL
LIN {X 0,Y 172.974,Z 572.339,A -85,B 0,C 180,E1 9422.079,E2 9422.079} C_VEL
LIN {X 0,Y 180.016,Z 564.435,A -85,B 0,C 180,E1 9416.258,E2 9416.258} C_VEL
LIN {X 0,Y 188.134,Z 554.944,A -85,B 0,C 180,E1 9411.16,E2 9411.16} C_VEL
LIN {X 0,Y 196.952,Z 543.894,A -85,B 0,C 180,E1 9406.735,E2 9406.735} C_VEL
LIN {X 0,Y 206.165,Z 531.271,A -85,B 0,C 180,E1 9402.916,E2 9402.916} C_VEL
LIN {X 0,Y 210.076,Z 525.372,A -85,B 0,C 180,E1 9401.421,E2 9401.421} C_VEL
LIN {X 0,Y 198.547,Z 528.942,A -85,B 0,C 180,E1 9398.643,E2 9398.643} C_VEL
LIN {X 0,Y 189.452,Z 531.492,A -85,B 0,C 180,E1 9395.862,E2 9395.862} C_VEL
LIN {X 0,Y 182.402,Z 533.361,A -85,B 0,C 180,E1 9393.242,E2 9393.242} C_VEL
LIN {X 0,Y 176.563,Z 534.828,A -85,B 0,C 180,E1 9390.642,E2 9390.642} C_VEL
LIN {X 0,Y 175.03,Z 535.113,A -85,B 0,C 180,E1 9389.802,E2 9389.802} C_VEL
LIN {X 0,Y 171.322,Z 536.047,A -85,B 0,C 180,E1 9387.833,E2 9387.833} C_VEL
LIN {X 0,Y 170.052,Z 536.197,A -85,B 0,C 180,E1 9386.92,E2 9386.92} C_VEL
LIN {X 0,Y 167.079,Z 537.032,A -85,B 0,C 180,E1 9385.144,E2 9385.144} C_VEL
LIN {X 0,Y 166.137,Z 537.024,A -85,B 0,C 180,E1 9383.969,E2 9383.969} C_VEL
LIN {X 0,Y 163.597,Z 549.318,A -85,B 0,C 180,E1 9378.901,E2 9378.901} C_VEL
LIN {X 0,Y 161.885,Z 559.867,A -85,B 0,C 180,E1 9373.575,E2 9373.575} C_VEL
LIN {X 0,Y 160.951,Z 569.046,A -85,B 0,C 180,E1 9367.856,E2 9367.856} C_VEL
LIN {X 0,Y 160.74,Z 576.359,A -85,B 0,C 180,E1 9362.14,E2 9362.14} C_VEL
LIN {X 0,Y 161.137,Z 582.094,A -85,B 0,C 180,E1 9356.443,E2 9356.443} C_VEL
LIN {X 0,Y 162.13,Z 586.006,A -85,B 0,C 180,E1 9351.543,E2 9351.543} C_VEL
LIN {X 0,Y 162.027,Z 587.769,A -85,B 0,C 180,E1 9348.871,E2 9348.871} C_VEL
LIN {X 0,Y 159.704,Z 591.334,A -85,B 0,C 180,E1 9341.441,E2 9341.441} C_VEL
LIN {X 0,Y 160.746,Z 592.184,A -85,B 0,C 180,E1 9339.103,E2 9339.103} C_VEL
LIN {X 0,Y 168.343,Z 593.83,A -85,B 0,C 180,E1 9332.018,E2 9332.018} C_VEL
LIN {X 0,Y 178.675,Z 593.716,A -85,B 0,C 180,E1 9325.585,E2 9325.585} C_VEL
LIN {X 0,Y 191.995,Z 591.843,A -85,B 0,C 180,E1 9319.778,E2 9319.778} C_VEL
LIN {X 0,Y 193.003,Z 591.662,A -85,B 0,C 180,E1 9319.36,E2 9319.36} C_VEL
LIN {X 0,Y 176.902,Z 597.798,A -85,B 0,C 180,E1 9312.709,E2 9312.709} C_VEL
LIN {X 0,Y 164.742,Z 602.421,A -85,B 0,C 180,E1 9304.788,E2 9304.788} C_VEL
LIN {X 0,Y 156.977,Z 605.261,A -85,B 0,C 180,E1 9296.074,E2 9296.074} C_VEL
LIN {X 0,Y 153.489,Z 606.36,A -85,B 0,C 180,E1 9287.831,E2 9287.831} C_VEL
LIN {X 0,Y 152.459,Z 609.889,A -85,B 0,C 180,E1 9280.202,E2 9280.202} C_VEL
LIN {X 0,Y 152.749,Z 611.487,A -85,B 0,C 180,E1 9273.756,E2 9273.756} C_VEL
LIN {X 0,Y 152.894,Z 611.681,A -85,B 0,C 180,E1 9268.878,E2 9268.878} C_VEL
LIN {X 0,Y 152.581,Z 610.959,A -85,B 0,C 180,E1 9263.606,E2 9263.606} C_VEL
LIN {X 0,Y 152.596,Z 608.67,A -85,B 0,C 180,E1 9256.745,E2 9256.745} C_VEL
LIN {X 0,Y 154.118,Z 604.634,A -85,B 0,C 180,E1 9249.495,E2 9249.495} C_VEL
LIN {X 0,Y 157.814,Z 598.497,A -85,B 0,C 180,E1 9242.044,E2 9242.044} C_VEL
LIN {X 0,Y 163.767,Z 590.311,A -85,B 0,C 180,E1 9234.98,E2 9234.98} C_VEL
LIN {X 0,Y 171.438,Z 580.472,A -85,B 0,C 180,E1 9228.777,E2 9228.777} C_VEL
LIN {X 0,Y 180.346,Z 569.031,A -85,B 0,C 180,E1 9223.428,E2 9223.428} C_VEL
LIN {X 0,Y 190.068,Z 556.008,A -85,B 0,C 180,E1 9218.875,E2 9218.875} C_VEL
LIN {X 0,Y 200.21,Z 541.347,A -85,B 0,C 180,E1 9215.017,E2 9215.017} C_VEL
LIN {X 0,Y 210.155,Z 525.522,A -85,B 0,C 180,E1 9211.877,E2 9211.877} C_VEL
LIN {X 0,Y 219.584,Z 508.568,A -85,B 0,C 180,E1 9209.314,E2 9209.314} C_VEL
LIN {X 0,Y 228.291,Z 490.517,A -85,B 0,C 180,E1 9207.245,E2 9207.245} C_VEL
LIN {X 0,Y 236.118,Z 471.305,A -85,B 0,C 180,E1 9205.587,E2 9205.587} C_VEL
LIN {X 0,Y 242.652,Z 451.643,A -85,B 0,C 180,E1 9204.333,E2 9204.333} C_VEL
LIN {X 0,Y 247.911,Z 431.224,A -85,B 0,C 180,E1 9203.401,E2 9203.401} C_VEL
LIN {X 0,Y 251.658,Z 410.109,A -85,B 0,C 180,E1 9202.707,E2 9202.707} C_VEL
LIN {X 0,Y 263.707,Z 285.061,A -85,B 0,C 180,E1 9199.887,E2 9199.887} C_VEL
LIN {X 0,Y 259.159,Z 275.272,A -85,B 0,C 180,E1 9196.531,E2 9196.531} C_VEL
LIN {X 0,Y 255.204,Z 267.49,A -85,B 0,C 180,E1 9193.019,E2 9193.019} C_VEL
LIN {X 0,Y 252.487,Z 262.375,A -85,B 0,C 180,E1 9190.034,E2 9190.034} C_VEL
LIN {X 0,Y 250.244,Z 258.418,A -85,B 0,C 180,E1 9186.884,E2 9186.884} C_VEL
LIN {X 0,Y 248.156,Z 254.462,A -85,B 0,C 180,E1 9182.294,E2 9182.294} C_VEL
LIN {X 0,Y 247.275,Z 253.696,A -85,B 0,C 180,E1 9176.754,E2 9176.754} C_VEL
LIN {X 0,Y 248.035,Z 254.635,A -85,B 0,C 180,E1 9172.355,E2 9172.355} C_VEL
LIN {X 0,Y 250.179,Z 259.006,A -85,B 0,C 180,E1 9167.536,E2 9167.536} C_VEL
LIN {X 0,Y 252.14,Z 262.751,A -85,B 0,C 180,E1 9164.709,E2 9164.709} C_VEL
LIN {X 0,Y 255.025,Z 268.335,A -85,B 0,C 180,E1 9161.483,E2 9161.483} C_VEL
LIN {X 0,Y 258.53,Z 275.562,A -85,B 0,C 180,E1 9158.324,E2 9158.324} C_VEL
LIN {X 0,Y 262.534,Z 284.437,A -85,B 0,C 180,E1 9155.292,E2 9155.292} C_VEL
LIN {X 0,Y 263.137,Z 286.286,A -85,B 0,C 180,E1 9154.843,E2 9154.843} C_VEL
LIN {X 0,Y 252.654,Z 402.022,A -85,B 0,C 180,E1 9152.352,E2 9152.352} C_VEL
LIN {X 0,Y 249.325,Z 421.98,A -85,B 0,C 180,E1 9151.654,E2 9151.654} C_VEL
LIN {X 0,Y 244.777,Z 440.862,A -85,B 0,C 180,E1 9150.7,E2 9150.7} C_VEL
LIN {X 0,Y 238.739,Z 459.884,A -85,B 0,C 180,E1 9149.386,E2 9149.386} C_VEL
LIN {X 0,Y 231.687,Z 477.691,A -85,B 0,C 180,E1 9147.76,E2 9147.76} C_VEL
LIN {X 0,Y 223.729,Z 494.437,A -85,B 0,C 180,E1 9145.765,E2 9145.765} C_VEL
LIN {X 0,Y 214.664,Z 510.718,A -85,B 0,C 180,E1 9143.236,E2 9143.236} C_VEL
LIN {X 0,Y 205.357,Z 525.25,A -85,B 0,C 180,E1 9140.286,E2 9140.286} C_VEL
LIN {X 0,Y 195.997,Z 538.228,A -85,B 0,C 180,E1 9136.841,E2 9136.841} C_VEL
LIN {X 0,Y 186.266,Z 550.418,A -85,B 0,C 180,E1 9132.557,E2 9132.557} C_VEL
LIN {X 0,Y 177.118,Z 560.916,A -85,B 0,C 180,E1 9127.563,E2 9127.563} C_VEL
LIN {X 0,Y 168.932,Z 569.731,A -85,B 0,C 180,E1 9121.784,E2 9121.784} C_VEL
LIN {X 0,Y 162.429,Z 576.544,A -85,B 0,C 180,E1 9115.522,E2 9115.522} C_VEL
LIN {X 0,Y 157.497,Z 581.751,A -85,B 0,C 180,E1 9108.504,E2 9108.504} C_VEL
LIN {X 0,Y 154.527,Z 585.122,A -85,B 0,C 180,E1 9101.19,E2 9101.19} C_VEL
LIN {X 0,Y 153.257,Z 586.779,A -85,B 0,C 180,E1 9093.738,E2 9093.738} C_VEL
LIN {X 0,Y 153.207,Z 586.827,A -85,B 0,C 180,E1 9086.883,E2 9086.883} C_VEL
LIN {X 0,Y 154.218,Z 585.486,A -85,B 0,C 180,E1 9079.916,E2 9079.916} C_VEL
LIN {X 0,Y 156.891,Z 582.419,A -85,B 0,C 180,E1 9072.568,E2 9072.568} C_VEL
LIN {X 0,Y 161.501,Z 577.531,A -85,B 0,C 180,E1 9065.491,E2 9065.491} C_VEL
LIN {X 0,Y 167.745,Z 571.033,A -85,B 0,C 180,E1 9059.131,E2 9059.131} C_VEL
LIN {X 0,Y 175.175,Z 563.116,A -85,B 0,C 180,E1 9053.584,E2 9053.584} C_VEL
LIN {X 0,Y 184.03,Z 553.155,A -85,B 0,C 180,E1 9048.481,E2 9048.481} C_VEL
LIN {X 0,Y 193.513,Z 541.582,A -85,B 0,C 180,E1 9044.092,E2 9044.092} C_VEL
LIN {X 0,Y 200.272,Z 532.652,A -85,B 0,C 180,E1 9041.416,E2 9041.416} C_VEL
LIN {X 0,Y 185.858,Z 536.526,A -85,B 0,C 180,E1 9037.439,E2 9037.439} C_VEL
LIN {X 0,Y 177.913,Z 538.479,A -85,B 0,C 180,E1 9034.585,E2 9034.585} C_VEL
LIN {X 0,Y 171.333,Z 539.994,A -85,B 0,C 180,E1 9031.684,E2 9031.684} C_VEL
LIN {X 0,Y 165.937,Z 541.202,A -85,B 0,C 180,E1 9028.82,E2 9028.82} C_VEL
LIN {X 0,Y 161.201,Z 542.214,A -85,B 0,C 180,E1 9025.734,E2 9025.734} C_VEL
LIN {X 0,Y 160.507,Z 542.235,A -85,B 0,C 180,E1 9025.063,E2 9025.063} C_VEL
LIN {X 0,Y 157.735,Z 543.049,A -85,B 0,C 180,E1 9023.143,E2 9023.143} C_VEL
LIN {X 0,Y 156.829,Z 543.019,A -85,B 0,C 180,E1 9021.801,E2 9021.801} C_VEL
LIN {X 0,Y 154.572,Z 554.913,A -85,B 0,C 180,E1 9016.151,E2 9016.151} C_VEL
LIN {X 0,Y 153.295,Z 564.57,A -85,B 0,C 180,E1 9010.524,E2 9010.524} C_VEL
LIN {X 0,Y 152.771,Z 572.93,A -85,B 0,C 180,E1 9004.505,E2 9004.505} C_VEL
LIN {X 0,Y 152.969,Z 579.931,A -85,B 0,C 180,E1 8998.128,E2 8998.128} C_VEL
LIN {X 0,Y 154.234,Z 585.845,A -85,B 0,C 180,E1 8991.05,E2 8991.05} C_VEL
LIN {X 0,Y 157.396,Z 590.194,A -85,B 0,C 180,E1 8983.77,E2 8983.77} C_VEL
LIN {X 0,Y 160.746,Z 592.184,A -85,B 0,C 180,E1 8979.103,E2 8979.103} C_VEL
LIN {X 0,Y 162.186,Z 593.076,A -85,B 0,C 180,E1 8976.412,E2 8976.412} C_VEL
LIN {X 0,Y 164.397,Z 594.847,A -85,B 0,C 180,E1 8969.221,E2 8969.221} C_VEL
LIN {X 0,Y 167.073,Z 595.114,A -85,B 0,C 180,E1 8966.914,E2 8966.914} C_VEL
LIN {X 0,Y 179.802,Z 594.604,A -85,B 0,C 180,E1 8960.659,E2 8960.659} C_VEL
LIN {X 0,Y 182.64,Z 594.326,A -85,B 0,C 180,E1 8959.432,E2 8959.432} C_VEL
LIN {X 0,Y 166.63,Z 599.44,A -85,B 0,C 180,E1 8952.228,E2 8952.228} C_VEL
LIN {X 0,Y 154.579,Z 603.098,A -85,B 0,C 180,E1 8943.356,E2 8943.356} C_VEL
LIN {X 0,Y 147.503,Z 604.837,A -85,B 0,C 180,E1 8933.577,E2 8933.577} C_VEL
LIN {X 0,Y 145.989,Z 605.245,A -85,B 0,C 180,E1 8929.611,E2 8929.611} C_VEL
LIN {X 0,Y 144.509,Z 608.971,A -85,B 0,C 180,E1 8921.578,E2 8921.578} C_VEL
LIN {X 0,Y 144.702,Z 610.719,A -85,B 0,C 180,E1 8914.759,E2 8914.759} C_VEL
LIN {X 0,Y 144.938,Z 611.086,A -85,B 0,C 180,E1 8909.607,E2 8909.607} C_VEL
LIN {X 0,Y 144.629,Z 610.469,A -85,B 0,C 180,E1 8904.05,E2 8904.05} C_VEL
LIN {X 0,Y 144.565,Z 608.541,A -85,B 0,C 180,E1 8897.211,E2 8897.211} C_VEL
LIN {X 0,Y 146.165,Z 604.478,A -85,B 0,C 180,E1 8889.166,E2 8889.166} C_VEL
LIN {X 0,Y 149.794,Z 598.836,A -85,B 0,C 180,E1 8881.714,E2 8881.714} C_VEL
LIN {X 0,Y 155.572,Z 591.393,A -85,B 0,C 180,E1 8874.663,E2 8874.663} C_VEL
LIN {X 0,Y 163.035,Z 582.422,A -85,B 0,C 180,E1 8868.434,E2 8868.434} C_VEL
LIN {X 0,Y 172.169,Z 571.442,A -85,B 0,C 180,E1 8862.801,E2 8862.801} C_VEL
LIN {X 0,Y 181.872,Z 559.31,A -85,B 0,C 180,E1 8858.176,E2 8858.176} C_VEL
LIN {X 0,Y 191.52,Z 546.369,A -85,B 0,C 180,E1 8854.429,E2 8854.429} C_VEL
LIN {X 0,Y 201.231,Z 532.176,A -85,B 0,C 180,E1 8851.287,E2 8851.287} C_VEL
LIN {X 0,Y 210.929,Z 516.344,A -85,B 0,C 180,E1 8848.604,E2 8848.604} C_VEL
LIN {X 0,Y 220.348,Z 498.737,A -85,B 0,C 180,E1 8846.343,E2 8846.343} C_VEL
LIN {X 0,Y 228.677,Z 480.493,A -85,B 0,C 180,E1 8844.575,E2 8844.575} C_VEL
LIN {X 0,Y 236.007,Z 461.171,A -85,B 0,C 180,E1 8843.176,E2 8843.176} C_VEL
LIN {X 0,Y 242.05,Z 441.153,A -85,B 0,C 180,E1 8842.119,E2 8842.119} C_VEL
LIN {X 0,Y 246.711,Z 420.235,A -85,B 0,C 180,E1 8841.335,E2 8841.335} C_VEL
LIN {X 0,Y 249.68,Z 398.846,A -85,B 0,C 180,E1 8840.756,E2 8840.756} C_VEL
LIN {X 0,Y 260.301,Z 289.473,A -85,B 0,C 180,E1 8838.359,E2 8838.359} C_VEL
LIN {X 0,Y 256.78,Z 281.608,A -85,B 0,C 180,E1 8835.527,E2 8835.527} C_VEL
LIN {X 0,Y 253.345,Z 274.513,A -85,B 0,C 180,E1 8832.247,E2 8832.247} C_VEL
LIN {X 0,Y 250.838,Z 269.632,A -85,B 0,C 180,E1 8829.29,E2 8829.29} C_VEL
LIN {X 0,Y 248.962,Z 266.115,A -85,B 0,C 180,E1 8826.456,E2 8826.456} C_VEL
LIN {X 0,Y 247.02,Z 262.288,A -85,B 0,C 180,E1 8821.855,E2 8821.855} C_VEL
LIN {X 0,Y 246.313,Z 261.656,A -85,B 0,C 180,E1 8816.437,E2 8816.437} C_VEL
LIN {X 0,Y 246.989,Z 262.537,A -85,B 0,C 180,E1 8812.556,E2 8812.556} C_VEL
LIN {X 0,Y 248.988,Z 266.855,A -85,B 0,C 180,E1 8807.829,E2 8807.829} C_VEL
LIN {X 0,Y 250.801,Z 270.5,A -85,B 0,C 180,E1 8805.099,E2 8805.099} C_VEL
LIN {X 0,Y 253.54,Z 276.019,A -85,B 0,C 180,E1 8801.907,E2 8801.907} C_VEL
LIN {X 0,Y 257.569,Z 284.89,A -85,B 0,C 180,E1 8798.179,E2 8798.179} C_VEL
LIN {X 0,Y 259.802,Z 290.39,A -85,B 0,C 180,E1 8796.39,E2 8796.39} C_VEL
LIN {X 0,Y 249.328,Z 402.32,A -85,B 0,C 180,E1 8794.012,E2 8794.012} C_VEL
LIN {X 0,Y 245.885,Z 422.382,A -85,B 0,C 180,E1 8793.323,E2 8793.323} C_VEL
LIN {X 0,Y 241.191,Z 441.332,A -85,B 0,C 180,E1 8792.384,E2 8792.384} C_VEL
LIN {X 0,Y 235.18,Z 459.805,A -85,B 0,C 180,E1 8791.136,E2 8791.136} C_VEL
LIN {X 0,Y 227.921,Z 477.705,A -85,B 0,C 180,E1 8789.54,E2 8789.54} C_VEL
LIN {X 0,Y 219.712,Z 494.526,A -85,B 0,C 180,E1 8787.579,E2 8787.579} C_VEL
LIN {X 0,Y 210.691,Z 510.293,A -85,B 0,C 180,E1 8785.181,E2 8785.181} C_VEL
LIN {X 0,Y 201.014,Z 524.984,A -85,B 0,C 180,E1 8782.264,E2 8782.264} C_VEL
LIN {X 0,Y 191.236,Z 538.099,A -85,B 0,C 180,E1 8778.838,E2 8778.838} C_VEL
LIN {X 0,Y 181.583,Z 549.739,A -85,B 0,C 180,E1 8774.811,E2 8774.811} C_VEL
LIN {X 0,Y 172.334,Z 559.938,A -85,B 0,C 180,E1 8770.088,E2 8770.088} C_VEL
LIN {X 0,Y 163.843,Z 568.669,A -85,B 0,C 180,E1 8764.576,E2 8764.576} C_VEL
LIN {X 0,Y 156.53,Z 575.876,A -85,B 0,C 180,E1 8758.206,E2 8758.206} C_VEL
LIN {X 0,Y 151.042,Z 581.234,A -85,B 0,C 180,E1 8751.349,E2 8751.349} C_VEL
LIN {X 0,Y 147.305,Z 585.046,A -85,B 0,C 180,E1 8743.74,E2 8743.74} C_VEL
LIN {X 0,Y 145.489,Z 587.116,A -85,B 0,C 180,E1 8735.914,E2 8735.914} C_VEL
LIN {X 0,Y 145.164,Z 587.56,A -85,B 0,C 180,E1 8728.419,E2 8728.419} C_VEL
LIN {X 0,Y 145.916,Z 586.658,A -85,B 0,C 180,E1 8721.327,E2 8721.327} C_VEL
LIN {X 0,Y 148.352,Z 584.035,A -85,B 0,C 180,E1 8713.554,E2 8713.554} C_VEL
LIN {X 0,Y 152.795,Z 579.618,A -85,B 0,C 180,E1 8706.062,E2 8706.062} C_VEL
LIN {X 0,Y 158.956,Z 573.648,A -85,B 0,C 180,E1 8699.367,E2 8699.367} C_VEL
LIN {X 0,Y 166.901,Z 565.754,A -85,B 0,C 180,E1 8693.194,E2 8693.194} C_VEL
LIN {X 0,Y 175.927,Z 556.279,A -85,B 0,C 180,E1 8687.881,E2 8687.881} C_VEL
LIN {X 0,Y 185.61,Z 545.253,A -85,B 0,C 180,E1 8683.343,E2 8683.343} C_VEL
LIN {X 0,Y 190.386,Z 539.291,A -85,B 0,C 180,E1 8681.332,E2 8681.332} C_VEL
LIN {X 0,Y 181.611,Z 541.497,A -85,B 0,C 180,E1 8678.876,E2 8678.876} C_VEL
LIN {X 0,Y 173.397,Z 543.397,A -85,B 0,C 180,E1 8676.028,E2 8676.028} C_VEL
LIN {X 0,Y 166.558,Z 544.884,A -85,B 0,C 180,E1 8673.113,E2 8673.113} C_VEL
LIN {X 0,Y 160.45,Z 546.138,A -85,B 0,C 180,E1 8669.903,E2 8669.903} C_VEL
LIN {X 0,Y 155.924,Z 547.111,A -85,B 0,C 180,E1 8667.084,E2 8667.084} C_VEL
LIN {X 0,Y 154.132,Z 547.464,A -85,B 0,C 180,E1 8665.763,E2 8665.763} C_VEL
LIN {X 0,Y 151.302,Z 547.996,A -85,B 0,C 180,E1 8663.361,E2 8663.361} C_VEL
LIN {X 0,Y 150.104,Z 548.28,A -85,B 0,C 180,E1 8662.315,E2 8662.315} C_VEL
LIN {X 0,Y 147.992,Z 548.743,A -85,B 0,C 180,E1 8660.156,E2 8660.156} C_VEL
LIN {X 0,Y 147.627,Z 548.714,A -85,B 0,C 180,E1 8659.28,E2 8659.28} C_VEL
LIN {X 0,Y 145.773,Z 560.004,A -85,B 0,C 180,E1 8653.083,E2 8653.083} C_VEL
LIN {X 0,Y 144.906,Z 569.363,A -85,B 0,C 180,E1 8646.737,E2 8646.737} C_VEL
LIN {X 0,Y 144.84,Z 576.879,A -85,B 0,C 180,E1 8640.396,E2 8640.396} C_VEL
LIN {X 0,Y 145.583,Z 583.147,A -85,B 0,C 180,E1 8633.692,E2 8633.692} C_VEL
LIN {X 0,Y 147.915,Z 588.395,A -85,B 0,C 180,E1 8626.316,E2 8626.316} C_VEL
LIN {X 0,Y 152.875,Z 592.34,A -85,B 0,C 180,E1 8618.516,E2 8618.516} C_VEL
LIN {X 0,Y 160.912,Z 594.599,A -85,B 0,C 180,E1 8611.01,E2 8611.01} C_VEL
LIN {X 0,Y 167.073,Z 595.114,A -85,B 0,C 180,E1 8606.914,E2 8606.914} C_VEL
LIN {X 0,Y 169.168,Z 595.375,A -85,B 0,C 180,E1 8605.053,E2 8605.053} C_VEL
LIN {X 0,Y 169.866,Z 595.925,A -85,B 0,C 180,E1 8602.708,E2 8602.708} C_VEL
LIN {X 0,Y 168.988,Z 596.725,A -85,B 0,C 180,E1 8600.15,E2 8600.15} C_VEL
LIN {X 0,Y 166.69,Z 597.698,A -85,B 0,C 180,E1 8597.645,E2 8597.645} C_VEL
LIN {X 0,Y 163.525,Z 598.652,A -85,B 0,C 180,E1 8595.653,E2 8595.653} C_VEL
LIN {X 0,Y 149.84,Z 602.003,A -85,B 0,C 180,E1 8586.913,E2 8586.913} C_VEL
LIN {X 0,Y 141.423,Z 603.57,A -85,B 0,C 180,E1 8577.361,E2 8577.361} C_VEL
LIN {X 0,Y 138.811,Z 603.886,A -85,B 0,C 180,E1 8572,E2 8572} C_VEL
LIN {X 0,Y 136.634,Z 607.999,A -85,B 0,C 180,E1 8563.282,E2 8563.282} C_VEL
LIN {X 0,Y 136.66,Z 609.941,A -85,B 0,C 180,E1 8555.723,E2 8555.723} C_VEL
LIN {X 0,Y 136.973,Z 610.461,A -85,B 0,C 180,E1 8550.003,E2 8550.003} C_VEL
LIN {X 0,Y 136.65,Z 609.897,A -85,B 0,C 180,E1 8544.123,E2 8544.123} C_VEL
LIN {X 0,Y 136.604,Z 607.99,A -85,B 0,C 180,E1 8536.772,E2 8536.772} C_VEL
LIN {X 0,Y 138.363,Z 604.042,A -85,B 0,C 180,E1 8528.377,E2 8528.377} C_VEL
LIN {X 0,Y 142.304,Z 598.494,A -85,B 0,C 180,E1 8520.542,E2 8520.542} C_VEL
LIN {X 0,Y 148.507,Z 591.148,A -85,B 0,C 180,E1 8513.19,E2 8513.19} C_VEL
LIN {X 0,Y 156.839,Z 581.84,A -85,B 0,C 180,E1 8506.491,E2 8506.491} C_VEL
LIN {X 0,Y 166.457,Z 570.978,A -85,B 0,C 180,E1 8500.817,E2 8500.817} C_VEL
LIN {X 0,Y 177.28,Z 558.112,A -85,B 0,C 180,E1 8495.912,E2 8495.912} C_VEL
LIN {X 0,Y 187.685,Z 544.681,A -85,B 0,C 180,E1 8492.112,E2 8492.112} C_VEL
LIN {X 0,Y 197.958,Z 530.088,A -85,B 0,C 180,E1 8489.004,E2 8489.004} C_VEL
LIN {X 0,Y 207.742,Z 514.474,A -85,B 0,C 180,E1 8486.469,E2 8486.469} C_VEL
LIN {X 0,Y 216.849,Z 497.873,A -85,B 0,C 180,E1 8484.41,E2 8484.41} C_VEL
LIN {X 0,Y 225.414,Z 479.555,A -85,B 0,C 180,E1 8482.694,E2 8482.694} C_VEL
LIN {X 0,Y 232.931,Z 460.104,A -85,B 0,C 180,E1 8481.339,E2 8481.339} C_VEL
LIN {X 0,Y 239.124,Z 439.844,A -85,B 0,C 180,E1 8480.32,E2 8480.32} C_VEL
LIN {X 0,Y 243.798,Z 418.914,A -85,B 0,C 180,E1 8479.573,E2 8479.573} C_VEL
LIN {X 0,Y 246.767,Z 397.389,A -85,B 0,C 180,E1 8479.014,E2 8479.014} C_VEL
LIN {X 0,Y 257.05,Z 293.886,A -85,B 0,C 180,E1 8476.77,E2 8476.77} C_VEL
LIN {X 0,Y 253.797,Z 286.405,A -85,B 0,C 180,E1 8473.847,E2 8473.847} C_VEL
LIN {X 0,Y 250.692,Z 279.691,A -85,B 0,C 180,E1 8470.455,E2 8470.455} C_VEL
LIN {X 0,Y 247.963,Z 274.178,A -85,B 0,C 180,E1 8466.482,E2 8466.482} C_VEL
LIN {X 0,Y 245.96,Z 270.176,A -85,B 0,C 180,E1 8461.63,E2 8461.63} C_VEL
LIN {X 0,Y 245.346,Z 269.612,A -85,B 0,C 180,E1 8456.261,E2 8456.261} C_VEL
LIN {X 0,Y 245.969,Z 270.514,A -85,B 0,C 180,E1 8452.669,E2 8452.669} C_VEL
LIN {X 0,Y 247.742,Z 274.559,A -85,B 0,C 180,E1 8448.24,E2 8448.24} C_VEL
LIN {X 0,Y 249.466,Z 278.245,A -85,B 0,C 180,E1 8445.492,E2 8445.492} C_VEL
LIN {X 0,Y 252.057,Z 283.765,A -85,B 0,C 180,E1 8442.334,E2 8442.334} C_VEL
LIN {X 0,Y 255.702,Z 292.238,A -85,B 0,C 180,E1 8438.795,E2 8438.795} C_VEL
LIN {X 0,Y 256.631,Z 294.872,A -85,B 0,C 180,E1 8437.968,E2 8437.968} C_VEL
LIN {X 0,Y 246.216,Z 402.616,A -85,B 0,C 180,E1 8435.715,E2 8435.715} C_VEL
LIN {X 0,Y 242.685,Z 422.674,A -85,B 0,C 180,E1 8435.043,E2 8435.043} C_VEL
LIN {X 0,Y 237.819,Z 441.8,A -85,B 0,C 180,E1 8434.117,E2 8434.117} C_VEL
LIN {X 0,Y 231.451,Z 460.779,A -85,B 0,C 180,E1 8432.858,E2 8432.858} C_VEL
LIN {X 0,Y 223.994,Z 478.58,A -85,B 0,C 180,E1 8431.294,E2 8431.294} C_VEL
LIN {X 0,Y 215.169,Z 496.022,A -85,B 0,C 180,E1 8429.275,E2 8429.275} C_VEL
LIN {X 0,Y 205.51,Z 512.192,A -85,B 0,C 180,E1 8426.802,E2 8426.802} C_VEL
LIN {X 0,Y 195.531,Z 526.669,A -85,B 0,C 180,E1 8423.892,E2 8423.892} C_VEL
LIN {X 0,Y 185.416,Z 539.615,A -85,B 0,C 180,E1 8420.452,E2 8420.452} C_VEL
LIN {X 0,Y 174.794,Z 551.764,A -85,B 0,C 180,E1 8416.113,E2 8416.113} C_VEL
LIN {X 0,Y 164.686,Z 562.238,A -85,B 0,C 180,E1 8410.969,E2 8410.969} C_VEL
LIN {X 0,Y 155.51,Z 571.04,A -85,B 0,C 180,E1 8404.903,E2 8404.903} C_VEL
LIN {X 0,Y 148.101,Z 577.846,A -85,B 0,C 180,E1 8398.199,E2 8398.199} C_VEL
LIN {X 0,Y 142.378,Z 583.049,A -85,B 0,C 180,E1 8390.553,E2 8390.553} C_VEL
LIN {X 0,Y 138.863,Z 586.416,A -85,B 0,C 180,E1 8382.472,E2 8382.472} C_VEL
LIN {X 0,Y 137.37,Z 588.015,A -85,B 0,C 180,E1 8374.59,E2 8374.59} C_VEL
LIN {X 0,Y 137.245,Z 588.143,A -85,B 0,C 180,E1 8367.074,E2 8367.074} C_VEL
LIN {X 0,Y 138.391,Z 586.883,A -85,B 0,C 180,E1 8359.17,E2 8359.17} C_VEL
LIN {X 0,Y 141.46,Z 583.908,A -85,B 0,C 180,E1 8351.024,E2 8351.024} C_VEL
LIN {X 0,Y 146.839,Z 579.011,A -85,B 0,C 180,E1 8343.128,E2 8343.128} C_VEL
LIN {X 0,Y 154.146,Z 572.367,A -85,B 0,C 180,E1 8336.091,E2 8336.091} C_VEL
LIN {X 0,Y 163.043,Z 563.938,A -85,B 0,C 180,E1 8329.913,E2 8329.913} C_VEL
LIN {X 0,Y 172.931,Z 553.873,A -85,B 0,C 180,E1 8324.667,E2 8324.667} C_VEL
LIN {X 0,Y 180.432,Z 545.619,A -85,B 0,C 180,E1 8321.363,E2 8321.363} C_VEL
LIN {X 0,Y 168.874,Z 548.11,A -85,B 0,C 180,E1 8317.579,E2 8317.579} C_VEL
LIN {X 0,Y 161.77,Z 549.564,A -85,B 0,C 180,E1 8314.656,E2 8314.656} C_VEL
LIN {X 0,Y 154.891,Z 550.869,A -85,B 0,C 180,E1 8311.093,E2 8311.093} C_VEL
LIN {X 0,Y 150.194,Z 551.82,A -85,B 0,C 180,E1 8308.208,E2 8308.208} C_VEL
LIN {X 0,Y 145.365,Z 552.709,A -85,B 0,C 180,E1 8304.375,E2 8304.375} C_VEL
LIN {X 0,Y 141.902,Z 553.45,A -85,B 0,C 180,E1 8301.061,E2 8301.061} C_VEL
LIN {X 0,Y 140.98,Z 553.606,A -85,B 0,C 180,E1 8299.904,E2 8299.904} C_VEL
LIN {X 0,Y 139.003,Z 554.144,A -85,B 0,C 180,E1 8297.585,E2 8297.585} C_VEL
LIN {X 0,Y 138.587,Z 554.098,A -85,B 0,C 180,E1 8296.343,E2 8296.343} C_VEL
LIN {X 0,Y 137.273,Z 564.061,A -85,B 0,C 180,E1 8290.068,E2 8290.068} C_VEL
LIN {X 0,Y 136.823,Z 572.26,A -85,B 0,C 180,E1 8283.772,E2 8283.772} C_VEL
LIN {X 0,Y 137.112,Z 579.265,A -85,B 0,C 180,E1 8277.075,E2 8277.075} C_VEL
LIN {X 0,Y 138.581,Z 585.427,A -85,B 0,C 180,E1 8269.609,E2 8269.609} C_VEL
LIN {X 0,Y 142.414,Z 590.585,A -85,B 0,C 180,E1 8261.414,E2 8261.414} C_VEL
LIN {X 0,Y 149.336,Z 594.183,A -85,B 0,C 180,E1 8253.348,E2 8253.348} C_VEL
LIN {X 0,Y 159.838,Z 596.115,A -85,B 0,C 180,E1 8245.738,E2 8245.738} C_VEL
LIN {X 0,Y 172.365,Z 596.301,A -85,B 0,C 180,E1 8239.532,E2 8239.532} C_VEL
LIN {X 0,Y 163.525,Z 598.652,A -85,B 0,C 180,E1 8235.653,E2 8235.653} C_VEL
LIN {X 0,Y 158.045,Z 599.785,A -85,B 0,C 180,E1 8233.454,E2 8233.454} C_VEL
LIN {X 0,Y 143.872,Z 601.442,A -85,B 0,C 180,E1 8228.372,E2 8228.372} C_VEL
LIN {X 0,Y 139.818,Z 601.845,A -85,B 0,C 180,E1 8225.714,E2 8225.714} C_VEL
LIN {X 0,Y 131.782,Z 602.579,A -85,B 0,C 180,E1 8214.432,E2 8214.432} C_VEL
LIN {X 0,Y 128.952,Z 606.723,A -85,B 0,C 180,E1 8205.749,E2 8205.749} C_VEL
LIN {X 0,Y 128.585,Z 609.097,A -85,B 0,C 180,E1 8197.15,E2 8197.15} C_VEL
LIN {X 0,Y 128.973,Z 609.775,A -85,B 0,C 180,E1 8190.891,E2 8190.891} C_VEL
LIN {X 0,Y 128.727,Z 609.485,A -85,B 0,C 180,E1 8185.102,E2 8185.102} C_VEL
LIN {X 0,Y 128.572,Z 607.763,A -85,B 0,C 180,E1 8177.426,E2 8177.426} C_VEL
LIN {X 0,Y 130.134,Z 604.293,A -85,B 0,C 180,E1 8168.834,E2 8168.834} C_VEL
LIN {X 0,Y 134.311,Z 598.808,A -85,B 0,C 180,E1 8160.084,E2 8160.084} C_VEL
LIN {X 0,Y 140.74,Z 591.767,A -85,B 0,C 180,E1 8152.344,E2 8152.344} C_VEL
LIN {X 0,Y 148.885,Z 583.33,A -85,B 0,C 180,E1 8145.703,E2 8145.703} C_VEL
LIN {X 0,Y 158.766,Z 572.944,A -85,B 0,C 180,E1 8139.801,E2 8139.801} C_VEL
LIN {X 0,Y 169.496,Z 561.056,A -85,B 0,C 180,E1 8134.903,E2 8134.903} C_VEL
LIN {X 0,Y 180.542,Z 547.729,A -85,B 0,C 180,E1 8130.867,E2 8130.867} C_VEL
LIN {X 0,Y 191.682,Z 532.856,A -85,B 0,C 180,E1 8127.536,E2 8127.536} C_VEL
LIN {X 0,Y 201.825,Z 517.572,A -85,B 0,C 180,E1 8124.966,E2 8124.966} C_VEL
LIN {X 0,Y 211.541,Z 500.84,A -85,B 0,C 180,E1 8122.833,E2 8122.833} C_VEL
LIN {X 0,Y 220.287,Z 483.245,A -85,B 0,C 180,E1 8121.139,E2 8121.139} C_VEL
LIN {X 0,Y 227.95,Z 464.815,A -85,B 0,C 180,E1 8119.809,E2 8119.809} C_VEL
LIN {X 0,Y 234.444,Z 445.454,A -85,B 0,C 180,E1 8118.782,E2 8118.782} C_VEL
LIN {X 0,Y 239.601,Z 425.111,A -85,B 0,C 180,E1 8118.006,E2 8118.006} C_VEL
LIN {X 0,Y 243.1,Z 404.397,A -85,B 0,C 180,E1 8117.427,E2 8117.427} C_VEL
LIN {X 0,Y 253.993,Z 298.375,A -85,B 0,C 180,E1 8115.136,E2 8115.136} C_VEL
LIN {X 0,Y 250.625,Z 290.434,A -85,B 0,C 180,E1 8111.681,E2 8111.681} C_VEL
LIN {X 0,Y 248.216,Z 285.122,A -85,B 0,C 180,E1 8108.571,E2 8108.571} C_VEL
LIN {X 0,Y 246.439,Z 281.507,A -85,B 0,C 180,E1 8105.587,E2 8105.587} C_VEL
LIN {X 0,Y 244.904,Z 278.065,A -85,B 0,C 180,E1 8101.403,E2 8101.403} C_VEL
LIN {X 0,Y 244.36,Z 277.554,A -85,B 0,C 180,E1 8096.246,E2 8096.246} C_VEL
LIN {X 0,Y 244.907,Z 278.344,A -85,B 0,C 180,E1 8092.964,E2 8092.964} C_VEL
LIN {X 0,Y 246.574,Z 282.406,A -85,B 0,C 180,E1 8088.539,E2 8088.539} C_VEL
LIN {X 0,Y 248.157,Z 285.989,A -85,B 0,C 180,E1 8085.891,E2 8085.891} C_VEL
LIN {X 0,Y 250.593,Z 291.503,A -85,B 0,C 180,E1 8082.767,E2 8082.767} C_VEL
LIN {X 0,Y 253.667,Z 299.111,A -85,B 0,C 180,E1 8079.595,E2 8079.595} C_VEL
LIN {X 0,Y 243.328,Z 402.911,A -85,B 0,C 180,E1 8077.461,E2 8077.461} C_VEL
LIN {X 0,Y 239.682,Z 423.073,A -85,B 0,C 180,E1 8076.803,E2 8076.803} C_VEL
LIN {X 0,Y 234.671,Z 442.265,A -85,B 0,C 180,E1 8075.898,E2 8075.898} C_VEL
LIN {X 0,Y 228.209,Z 461.055,A -85,B 0,C 180,E1 8074.686,E2 8074.686} C_VEL
LIN {X 0,Y 220.284,Z 479.434,A -85,B 0,C 180,E1 8073.109,E2 8073.109} C_VEL
LIN {X 0,Y 211.209,Z 496.8,A -85,B 0,C 180,E1 8071.134,E2 8071.134} C_VEL
LIN {X 0,Y 201.718,Z 512.247,A -85,B 0,C 180,E1 8068.824,E2 8068.824} C_VEL
LIN {X 0,Y 191.652,Z 526.423,A -85,B 0,C 180,E1 8066.045,E2 8066.045} C_VEL
LIN {X 0,Y 180.67,Z 540.015,A -85,B 0,C 180,E1 8062.499,E2 8062.499} C_VEL
LIN {X 0,Y 169.928,Z 551.811,A -85,B 0,C 180,E1 8058.325,E2 8058.325} C_VEL
LIN {X 0,Y 159.271,Z 562.379,A -85,B 0,C 180,E1 8053.175,E2 8053.175} C_VEL
LIN {X 0,Y 149.466,Z 571.301,A -85,B 0,C 180,E1 8047.014,E2 8047.014} C_VEL
LIN {X 0,Y 141.075,Z 578.497,A -85,B 0,C 180,E1 8039.74,E2 8039.74} C_VEL
LIN {X 0,Y 134.897,Z 583.697,A -85,B 0,C 180,E1 8031.75,E2 8031.75} C_VEL
LIN {X 0,Y 131.061,Z 587.063,A -85,B 0,C 180,E1 8023.228,E2 8023.228} C_VEL
LIN {X 0,Y 129.388,Z 588.707,A -85,B 0,C 180,E1 8014.529,E2 8014.529} C_VEL
LIN {X 0,Y 129.278,Z 588.789,A -85,B 0,C 180,E1 8006.894,E2 8006.894} C_VEL
LIN {X 0,Y 130.545,Z 587.53,A -85,B 0,C 180,E1 7998.511,E2 7998.511} C_VEL
LIN {X 0,Y 133.903,Z 584.557,A -85,B 0,C 180,E1 7989.908,E2 7989.908} C_VEL
LIN {X 0,Y 139.654,Z 579.721,A -85,B 0,C 180,E1 7981.719,E2 7981.719} C_VEL
LIN {X 0,Y 147.549,Z 573.021,A -85,B 0,C 180,E1 7974.351,E2 7974.351} C_VEL
LIN {X 0,Y 156.988,Z 564.595,A -85,B 0,C 180,E1 7968.027,E2 7968.027} C_VEL
LIN {X 0,Y 167.39,Z 554.538,A -85,B 0,C 180,E1 7962.715,E2 7962.715} C_VEL
LIN {X 0,Y 170.397,Z 551.387,A -85,B 0,C 180,E1 7961.313,E2 7961.313} C_VEL
LIN {X 0,Y 156.99,Z 554.032,A -85,B 0,C 180,E1 7956.322,E2 7956.322} C_VEL
LIN {X 0,Y 144.858,Z 556.271,A -85,B 0,C 180,E1 7949.801,E2 7949.801} C_VEL
LIN {X 0,Y 135.734,Z 557.954,A -85,B 0,C 180,E1 7942.067,E2 7942.067} C_VEL
LIN {X 0,Y 132.466,Z 558.663,A -85,B 0,C 180,E1 7937.993,E2 7937.993} C_VEL
LIN {X 0,Y 131.703,Z 558.832,A -85,B 0,C 180,E1 7936.768,E2 7936.768} C_VEL
LIN {X 0,Y 129.911,Z 559.376,A -85,B 0,C 180,E1 7933.804,E2 7933.804} C_VEL
LIN {X 0,Y 129.726,Z 559.51,A -85,B 0,C 180,E1 7932.69,E2 7932.69} C_VEL
LIN {X 0,Y 128.935,Z 568.86,A -85,B 0,C 180,E1 7925.787,E2 7925.787} C_VEL
LIN {X 0,Y 129.007,Z 576.318,A -85,B 0,C 180,E1 7918.991,E2 7918.991} C_VEL
LIN {X 0,Y 130.028,Z 582.856,A -85,B 0,C 180,E1 7911.6,E2 7911.6} C_VEL
LIN {X 0,Y 133.26,Z 588.873,A -85,B 0,C 180,E1 7902.986,E2 7902.986} C_VEL
LIN {X 0,Y 139.49,Z 593.345,A -85,B 0,C 180,E1 7894.528,E2 7894.528} C_VEL
LIN {X 0,Y 149.103,Z 596.263,A -85,B 0,C 180,E1 7886.642,E2 7886.642} C_VEL
LIN {X 0,Y 162.131,Z 597.551,A -85,B 0,C 180,E1 7879.645,E2 7879.645} C_VEL
LIN {X 0,Y 146.24,Z 600.802,A -85,B 0,C 180,E1 7871.026,E2 7871.026} C_VEL
LIN {X 0,Y 139.818,Z 601.845,A -85,B 0,C 180,E1 7865.714,E2 7865.714} C_VEL
LIN {X 0,Y 137.015,Z 602.029,A -85,B 0,C 180,E1 7863.866,E2 7863.866} C_VEL
LIN {X 0,Y 126.771,Z 601.152,A -85,B 0,C 180,E1 7858.983,E2 7858.983} C_VEL
LIN {X 0,Y 125.221,Z 601.041,A -85,B 0,C 180,E1 7857.466,E2 7857.466} C_VEL
LIN {X 0,Y 121.322,Z 605.705,A -85,B 0,C 180,E1 7847.757,E2 7847.757} C_VEL
LIN {X 0,Y 120.558,Z 608.361,A -85,B 0,C 180,E1 7838.108,E2 7838.108} C_VEL
LIN {X 0,Y 120.949,Z 609.075,A -85,B 0,C 180,E1 7831.898,E2 7831.898} C_VEL
LIN {X 0,Y 120.893,Z 609.013,A -85,B 0,C 180,E1 7827.159,E2 7827.159} C_VEL
LIN {X 0,Y 120.515,Z 608.011,A -85,B 0,C 180,E1 7819.969,E2 7819.969} C_VEL
LIN {X 0,Y 121.533,Z 605.12,A -85,B 0,C 180,E1 7810.79,E2 7810.79} C_VEL
LIN {X 0,Y 124.986,Z 600.563,A -85,B 0,C 180,E1 7801.84,E2 7801.84} C_VEL
LIN {X 0,Y 131.01,Z 594.273,A -85,B 0,C 180,E1 7793.47,E2 7793.47} C_VEL
LIN {X 0,Y 139.787,Z 585.775,A -85,B 0,C 180,E1 7785.664,E2 7785.664} C_VEL
LIN {X 0,Y 149.945,Z 575.872,A -85,B 0,C 180,E1 7779.306,E2 7779.306} C_VEL
LIN {X 0,Y 160.769,Z 564.763,A -85,B 0,C 180,E1 7774.197,E2 7774.197} C_VEL
LIN {X 0,Y 172.098,Z 552.168,A -85,B 0,C 180,E1 7769.976,E2 7769.976} C_VEL
LIN {X 0,Y 183.336,Z 538.36,A -85,B 0,C 180,E1 7766.564,E2 7766.564} C_VEL
LIN {X 0,Y 194.432,Z 523.023,A -85,B 0,C 180,E1 7763.749,E2 7763.749} C_VEL
LIN {X 0,Y 205.144,Z 506.005,A -85,B 0,C 180,E1 7761.427,E2 7761.427} C_VEL
LIN {X 0,Y 214.944,Z 487.73,A -85,B 0,C 180,E1 7759.581,E2 7759.581} C_VEL
LIN {X 0,Y 223.137,Z 469.472,A -85,B 0,C 180,E1 7758.21,E2 7758.21} C_VEL
LIN {X 0,Y 230.187,Z 450.1,A -85,B 0,C 180,E1 7757.143,E2 7757.143} C_VEL
LIN {X 0,Y 235.939,Z 429.491,A -85,B 0,C 180,E1 7756.331,E2 7756.331} C_VEL
LIN {X 0,Y 239.993,Z 408.245,A -85,B 0,C 180,E1 7755.721,E2 7755.721} C_VEL
LIN {X 0,Y 251.184,Z 303.237,A -85,B 0,C 180,E1 7753.53,E2 7753.53} C_VEL
LIN {X 0,Y 248.232,Z 296.001,A -85,B 0,C 180,E1 7750.091,E2 7750.091} C_VEL
LIN {X 0,Y 246.3,Z 291.647,A -85,B 0,C 180,E1 7747.229,E2 7747.229} C_VEL
LIN {X 0,Y 245.202,Z 289.202,A -85,B 0,C 180,E1 7745.146,E2 7745.146} C_VEL
LIN {X 0,Y 243.863,Z 285.956,A -85,B 0,C 180,E1 7741.174,E2 7741.174} C_VEL
LIN {X 0,Y 243.402,Z 285.521,A -85,B 0,C 180,E1 7735.995,E2 7735.995} C_VEL
LIN {X 0,Y 243.871,Z 286.249,A -85,B 0,C 180,E1 7733.171,E2 7733.171} C_VEL
LIN {X 0,Y 245.42,Z 290.251,A -85,B 0,C 180,E1 7728.841,E2 7728.841} C_VEL
LIN {X 0,Y 246.861,Z 293.731,A -85,B 0,C 180,E1 7726.293,E2 7726.293} C_VEL
LIN {X 0,Y 249.283,Z 299.622,A -85,B 0,C 180,E1 7723.034,E2 7723.034} C_VEL
LIN {X 0,Y 250.856,Z 303.998,A -85,B 0,C 180,E1 7721.235,E2 7721.235} C_VEL
LIN {X 0,Y 240.67,Z 403.205,A -85,B 0,C 180,E1 7719.247,E2 7719.247} C_VEL
LIN {X 0,Y 236.938,Z 423.364,A -85,B 0,C 180,E1 7718.61,E2 7718.61} C_VEL
LIN {X 0,Y 231.755,Z 442.729,A -85,B 0,C 180,E1 7717.726,E2 7717.726} C_VEL
LIN {X 0,Y 225.066,Z 461.671,A -85,B 0,C 180,E1 7716.541,E2 7716.541} C_VEL
LIN {X 0,Y 217.213,Z 479.466,A -85,B 0,C 180,E1 7715.064,E2 7715.064} C_VEL
LIN {X 0,Y 207.881,Z 496.92,A -85,B 0,C 180,E1 7713.147,E2 7713.147} C_VEL
LIN {X 0,Y 197.794,Z 512.859,A -85,B 0,C 180,E1 7710.824,E2 7710.824} C_VEL
LIN {X 0,Y 187.307,Z 527.142,A -85,B 0,C 180,E1 7708.072,E2 7708.072} C_VEL
LIN {X 0,Y 175.899,Z 540.723,A -85,B 0,C 180,E1 7704.563,E2 7704.563} C_VEL
LIN {X 0,Y 164.656,Z 552.544,A -85,B 0,C 180,E1 7700.386,E2 7700.386} C_VEL
LIN {X 0,Y 153.52,Z 563.045,A -85,B 0,C 180,E1 7695.224,E2 7695.224} C_VEL
LIN {X 0,Y 143.137,Z 571.957,A -85,B 0,C 180,E1 7688.949,E2 7688.949} C_VEL
LIN {X 0,Y 134.163,Z 579.148,A -85,B 0,C 180,E1 7681.441,E2 7681.441} C_VEL
LIN {X 0,Y 127.482,Z 584.346,A -85,B 0,C 180,E1 7673.085,E2 7673.085} C_VEL
LIN {X 0,Y 123.284,Z 587.71,A -85,B 0,C 180,E1 7664.079,E2 7664.079} C_VEL
LIN {X 0,Y 121.452,Z 589.329,A -85,B 0,C 180,E1 7655.028,E2 7655.028} C_VEL
LIN {X 0,Y 121.313,Z 589.434,A -85,B 0,C 180,E1 7646.69,E2 7646.69} C_VEL
LIN {X 0,Y 122.715,Z 588.177,A -85,B 0,C 180,E1 7637.767,E2 7637.767} C_VEL
LIN {X 0,Y 126.401,Z 585.206,A -85,B 0,C 180,E1 7628.659,E2 7628.659} C_VEL
LIN {X 0,Y 132.576,Z 580.419,A -85,B 0,C 180,E1 7620.145,E2 7620.145} C_VEL
LIN {X 0,Y 141.099,Z 573.673,A -85,B 0,C 180,E1 7612.45,E2 7612.45} C_VEL
LIN {X 0,Y 151.115,Z 565.251,A -85,B 0,C 180,E1 7605.991,E2 7605.991} C_VEL
LIN {X 0,Y 160.36,Z 556.718,A -85,B 0,C 180,E1 7601.252,E2 7601.252} C_VEL
LIN {X 0,Y 145.826,Z 559.382,A -85,B 0,C 180,E1 7595.167,E2 7595.167} C_VEL
LIN {X 0,Y 133.658,Z 561.465,A -85,B 0,C 180,E1 7587.151,E2 7587.151} C_VEL
LIN {X 0,Y 129.182,Z 562.263,A -85,B 0,C 180,E1 7582.769,E2 7582.769} C_VEL
LIN {X 0,Y 126.055,Z 562.955,A -85,B 0,C 180,E1 7578.979,E2 7578.979} C_VEL
LIN {X 0,Y 123.203,Z 563.687,A -85,B 0,C 180,E1 7574.092,E2 7574.092} C_VEL
LIN {X 0,Y 121.231,Z 564.457,A -85,B 0,C 180,E1 7569.495,E2 7569.495} C_VEL
LIN {X 0,Y 121.176,Z 564.669,A -85,B 0,C 180,E1 7568.303,E2 7568.303} C_VEL
LIN {X 0,Y 120.974,Z 573.096,A -85,B 0,C 180,E1 7560.948,E2 7560.948} C_VEL
LIN {X 0,Y 121.693,Z 580.114,A -85,B 0,C 180,E1 7553.396,E2 7553.396} C_VEL
LIN {X 0,Y 124.511,Z 586.991,A -85,B 0,C 180,E1 7544.156,E2 7544.156} C_VEL
LIN {X 0,Y 130.428,Z 592.323,A -85,B 0,C 180,E1 7535.063,E2 7535.063} C_VEL
LIN {X 0,Y 139.904,Z 596.111,A -85,B 0,C 180,E1 7526.614,E2 7526.614} C_VEL
LIN {X 0,Y 151.785,Z 598.21,A -85,B 0,C 180,E1 7519.65,E2 7519.65} C_VEL
LIN {X 0,Y 136.174,Z 600.463,A -85,B 0,C 180,E1 7510.255,E2 7510.255} C_VEL
LIN {X 0,Y 126.334,Z 601.028,A -85,B 0,C 180,E1 7499.389,E2 7499.389} C_VEL
LIN {X 0,Y 125.221,Z 601.041,A -85,B 0,C 180,E1 7497.466,E2 7497.466} C_VEL
LIN {X 0,Y 122.183,Z 603.013,A -85,B 0,C 180,E1 7493.99,E2 7493.99} C_VEL
LIN {X 0,Y 113.728,Z 606.315,A -85,B 0,C 180,E1 7485.237,E2 7485.237} C_VEL
LIN {X 0,Y 112.56,Z 607.163,A -85,B 0,C 180,E1 7481.653,E2 7481.653} C_VEL
LIN {X 0,Y 112.863,Z 608.34,A -85,B 0,C 180,E1 7473.559,E2 7473.559} C_VEL
LIN {X 0,Y 112.991,Z 608.452,A -85,B 0,C 180,E1 7468.482,E2 7468.482} C_VEL
LIN {X 0,Y 112.574,Z 607.775,A -85,B 0,C 180,E1 7461.833,E2 7461.833} C_VEL
LIN {X 0,Y 113.234,Z 605.359,A -85,B 0,C 180,E1 7452.002,E2 7452.002} C_VEL
LIN {X 0,Y 116.464,Z 601.287,A -85,B 0,C 180,E1 7442.384,E2 7442.384} C_VEL
LIN {X 0,Y 122.45,Z 595.487,A -85,B 0,C 180,E1 7433.414,E2 7433.414} C_VEL
LIN {X 0,Y 131.494,Z 587.38,A -85,B 0,C 180,E1 7425,E2 7425} C_VEL
LIN {X 0,Y 142.303,Z 577.612,A -85,B 0,C 180,E1 7418.104,E2 7418.104} C_VEL
LIN {X 0,Y 154.17,Z 566.24,A -85,B 0,C 180,E1 7412.535,E2 7412.535} C_VEL
LIN {X 0,Y 166.535,Z 553.278,A -85,B 0,C 180,E1 7408.051,E2 7408.051} C_VEL
LIN {X 0,Y 178.999,Z 538.667,A -85,B 0,C 180,E1 7404.433,E2 7404.433} C_VEL
LIN {X 0,Y 190.861,Z 522.859,A -85,B 0,C 180,E1 7401.593,E2 7401.593} C_VEL
LIN {X 0,Y 201.874,Z 505.915,A -85,B 0,C 180,E1 7399.355,E2 7399.355} C_VEL
LIN {X 0,Y 211.872,Z 487.817,A -85,B 0,C 180,E1 7397.591,E2 7397.591} C_VEL
LIN {X 0,Y 220.288,Z 469.535,A -85,B 0,C 180,E1 7396.273,E2 7396.273} C_VEL
LIN {X 0,Y 227.479,Z 450.277,A -85,B 0,C 180,E1 7395.257,E2 7395.257} C_VEL
LIN {X 0,Y 233.182,Z 430.449,A -85,B 0,C 180,E1 7394.506,E2 7394.506} C_VEL
LIN {X 0,Y 237.256,Z 410.229,A -85,B 0,C 180,E1 7393.937,E2 7393.937} C_VEL
LIN {X 0,Y 241.62,Z 372.79,A -85,B 0,C 180,E1 7393.147,E2 7393.147} C_VEL
LIN {X 0,Y 248.516,Z 308.104,A -85,B 0,C 180,E1 7391.84,E2 7391.84} C_VEL
LIN {X 0,Y 245.99,Z 301.57,A -85,B 0,C 180,E1 7388.414,E2 7388.414} C_VEL
LIN {X 0,Y 244.089,Z 297.084,A -85,B 0,C 180,E1 7384.934,E2 7384.934} C_VEL
LIN {X 0,Y 242.826,Z 293.849,A -85,B 0,C 180,E1 7380.943,E2 7380.943} C_VEL
LIN {X 0,Y 242.428,Z 293.465,A -85,B 0,C 180,E1 7375.979,E2 7375.979} C_VEL
LIN {X 0,Y 242.859,Z 294.255,A -85,B 0,C 180,E1 7373.261,E2 7373.261} C_VEL
LIN {X 0,Y 244.201,Z 297.939,A -85,B 0,C 180,E1 7369.275,E2 7369.275} C_VEL
LIN {X 0,Y 245.644,Z 301.645,A -85,B 0,C 180,E1 7366.584,E2 7366.584} C_VEL
LIN {X 0,Y 247.786,Z 307.328,A -85,B 0,C 180,E1 7363.532,E2 7363.532} C_VEL
LIN {X 0,Y 248.253,Z 308.931,A -85,B 0,C 180,E1 7362.915,E2 7362.915} C_VEL
LIN {X 0,Y 238.225,Z 403.66,A -85,B 0,C 180,E1 7361.066,E2 7361.066} C_VEL
LIN {X 0,Y 234.423,Z 423.703,A -85,B 0,C 180,E1 7360.455,E2 7360.455} C_VEL
LIN {X 0,Y 229.06,Z 443.256,A -85,B 0,C 180,E1 7359.595,E2 7359.595} C_VEL
LIN {X 0,Y 222.45,Z 461.6,A -85,B 0,C 180,E1 7358.494,E2 7358.494} C_VEL
LIN {X 0,Y 214.297,Z 479.696,A -85,B 0,C 180,E1 7357.054,E2 7357.054} C_VEL
LIN {X 0,Y 204.819,Z 497.028,A -85,B 0,C 180,E1 7355.224,E2 7355.224} C_VEL
LIN {X 0,Y 194.246,Z 513.297,A -85,B 0,C 180,E1 7352.931,E2 7352.931} C_VEL
LIN {X 0,Y 183.207,Z 527.857,A -85,B 0,C 180,E1 7350.193,E2 7350.193} C_VEL
LIN {X 0,Y 171.367,Z 541.429,A -85,B 0,C 180,E1 7346.738,E2 7346.738} C_VEL
LIN {X 0,Y 159.61,Z 553.274,A -85,B 0,C 180,E1 7342.579,E2 7342.579} C_VEL
LIN {X 0,Y 147.978,Z 563.709,A -85,B 0,C 180,E1 7337.429,E2 7337.429} C_VEL
LIN {X 0,Y 136.985,Z 572.613,A -85,B 0,C 180,E1 7331.061,E2 7331.061} C_VEL
LIN {X 0,Y 127.809,Z 579.502,A -85,B 0,C 180,E1 7323.737,E2 7323.737} C_VEL
LIN {X 0,Y 120.447,Z 584.795,A -85,B 0,C 180,E1 7315.044,E2 7315.044} C_VEL
LIN {X 0,Y 115.707,Z 588.238,A -85,B 0,C 180,E1 7305.535,E2 7305.535} C_VEL
LIN {X 0,Y 113.522,Z 589.953,A -85,B 0,C 180,E1 7295.556,E2 7295.556} C_VEL
LIN {X 0,Y 113.322,Z 590.099,A -85,B 0,C 180,E1 7286.962,E2 7286.962} C_VEL
LIN {X 0,Y 114.824,Z 588.89,A -85,B 0,C 180,E1 7277.235,E2 7277.235} C_VEL
LIN {X 0,Y 118.7,Z 586.048,A -85,B 0,C 180,E1 7267.722,E2 7267.722} C_VEL
LIN {X 0,Y 124.889,Z 581.646,A -85,B 0,C 180,E1 7259.174,E2 7259.174} C_VEL
LIN {X 0,Y 133.308,Z 575.491,A -85,B 0,C 180,E1 7251.496,E2 7251.496} C_VEL
LIN {X 0,Y 143.075,Z 567.897,A -85,B 0,C 180,E1 7245.101,E2 7245.101} C_VEL
LIN {X 0,Y 150.294,Z 561.73,A -85,B 0,C 180,E1 7241.254,E2 7241.254} C_VEL
LIN {X 0,Y 133.459,Z 564.487,A -85,B 0,C 180,E1 7232.952,E2 7232.952} C_VEL
LIN {X 0,Y 123.127,Z 566.224,A -85,B 0,C 180,E1 7224.467,E2 7224.467} C_VEL
LIN {X 0,Y 116.461,Z 567.691,A -85,B 0,C 180,E1 7214.926,E2 7214.926} C_VEL
LIN {X 0,Y 114.325,Z 568.497,A -85,B 0,C 180,E1 7209.566,E2 7209.566} C_VEL
LIN {X 0,Y 112.955,Z 569.44,A -85,B 0,C 180,E1 7204.062,E2 7204.062} C_VEL
LIN {X 0,Y 113.034,Z 569.506,A -85,B 0,C 180,E1 7203.043,E2 7203.043} C_VEL
LIN {X 0,Y 113.465,Z 576.856,A -85,B 0,C 180,E1 7195.452,E2 7195.452} C_VEL
LIN {X 0,Y 115.657,Z 584.283,A -85,B 0,C 180,E1 7185.993,E2 7185.993} C_VEL
LIN {X 0,Y 121.395,Z 590.829,A -85,B 0,C 180,E1 7175.682,E2 7175.682} C_VEL
LIN {X 0,Y 131.215,Z 595.654,A -85,B 0,C 180,E1 7166.203,E2 7166.203} C_VEL
LIN {X 0,Y 141.607,Z 598.229,A -85,B 0,C 180,E1 7159.695,E2 7159.695} C_VEL
LIN {X 0,Y 126.225,Z 599.515,A -85,B 0,C 180,E1 7149.327,E2 7149.327} C_VEL
LIN {X 0,Y 119.058,Z 599.464,A -85,B 0,C 180,E1 7140.82,E2 7140.82} C_VEL
LIN {X 0,Y 114.146,Z 604.326,A -85,B 0,C 180,E1 7131.051,E2 7131.051} C_VEL
LIN {X 0,Y 112.56,Z 607.163,A -85,B 0,C 180,E1 7121.653,E2 7121.653} C_VEL
LIN {X 0,Y 111.634,Z 607.87,A -85,B 0,C 180,E1 7118.011,E2 7118.011} C_VEL
LIN {X 0,Y 109.009,Z 608.213,A -85,B 0,C 180,E1 7113.257,E2 7113.257} C_VEL
LIN {X 0,Y 104.793,Z 607.577,A -85,B 0,C 180,E1 7104.326,E2 7104.326} C_VEL
LIN {X 0,Y 104.647,Z 607.399,A -85,B 0,C 180,E1 7103.079,E2 7103.079} C_VEL
LIN {X 0,Y 104.977,Z 605.518,A -85,B 0,C 180,E1 7093.401,E2 7093.401} C_VEL
LIN {X 0,Y 107.952,Z 601.834,A -85,B 0,C 180,E1 7083.014,E2 7083.014} C_VEL
LIN {X 0,Y 113.883,Z 596.462,A -85,B 0,C 180,E1 7073.347,E2 7073.347} C_VEL
LIN {X 0,Y 123.06,Z 588.868,A -85,B 0,C 180,E1 7064.362,E2 7064.362} C_VEL
LIN {X 0,Y 134.119,Z 579.645,A -85,B 0,C 180,E1 7057.096,E2 7057.096} C_VEL
LIN {X 0,Y 146.321,Z 568.823,A -85,B 0,C 180,E1 7051.287,E2 7051.287} C_VEL
LIN {X 0,Y 158.918,Z 556.568,A -85,B 0,C 180,E1 7046.7,E2 7046.7} C_VEL
LIN {X 0,Y 170.827,Z 543.678,A -85,B 0,C 180,E1 7043.236,E2 7043.236} C_VEL
LIN {X 0,Y 182.463,Z 529.516,A -85,B 0,C 180,E1 7040.446,E2 7040.446} C_VEL
LIN {X 0,Y 194.058,Z 513.307,A -85,B 0,C 180,E1 7038.089,E2 7038.089} C_VEL
LIN {X 0,Y 204.633,Z 496.052,A -85,B 0,C 180,E1 7036.243,E2 7036.243} C_VEL
LIN {X 0,Y 214.063,Z 477.733,A -85,B 0,C 180,E1 7034.798,E2 7034.798} C_VEL
LIN {X 0,Y 222.262,Z 458.225,A -85,B 0,C 180,E1 7033.675,E2 7033.675} C_VEL
LIN {X 0,Y 228.71,Z 438.759,A -85,B 0,C 180,E1 7032.875,E2 7032.875} C_VEL
LIN {X 0,Y 233.75,Z 417.902,A -85,B 0,C 180,E1 7032.253,E2 7032.253} C_VEL
LIN {X 0,Y 236.987,Z 396.437,A -85,B 0,C 180,E1 7031.768,E2 7031.768} C_VEL
LIN {X 0,Y 246.057,Z 313.216,A -85,B 0,C 180,E1 7030.129,E2 7030.129} C_VEL
LIN {X 0,Y 244.188,Z 308.017,A -85,B 0,C 180,E1 7027.174,E2 7027.174} C_VEL
LIN {X 0,Y 242.777,Z 304.591,A -85,B 0,C 180,E1 7024.251,E2 7024.251} C_VEL
LIN {X 0,Y 241.781,Z 301.742,A -85,B 0,C 180,E1 7020.71,E2 7020.71} C_VEL
LIN {X 0,Y 241.476,Z 301.439,A -85,B 0,C 180,E1 7015.725,E2 7015.725} C_VEL
LIN {X 0,Y 241.827,Z 302.167,A -85,B 0,C 180,E1 7013.471,E2 7013.471} C_VEL
LIN {X 0,Y 243.054,Z 305.795,A -85,B 0,C 180,E1 7009.571,E2 7009.571} C_VEL
LIN {X 0,Y 244.635,Z 310.095,A -85,B 0,C 180,E1 7006.528,E2 7006.528} C_VEL
LIN {X 0,Y 245.851,Z 313.873,A -85,B 0,C 180,E1 7004.63,E2 7004.63} C_VEL
LIN {X 0,Y 236.052,Z 403.952,A -85,B 0,C 180,E1 7002.925,E2 7002.925} C_VEL
LIN {X 0,Y 232.154,Z 424.052,A -85,B 0,C 180,E1 7002.338,E2 7002.338} C_VEL
LIN {X 0,Y 226.658,Z 443.652,A -85,B 0,C 180,E1 7001.514,E2 7001.514} C_VEL
LIN {X 0,Y 219.662,Z 462.56,A -85,B 0,C 180,E1 7000.422,E2 7000.422} C_VEL
LIN {X 0,Y 211.43,Z 480.35,A -85,B 0,C 180,E1 6999.058,E2 6999.058} C_VEL
LIN {X 0,Y 201.611,Z 497.816,A -85,B 0,C 180,E1 6997.28,E2 6997.28} C_VEL
LIN {X 0,Y 190.747,Z 514.034,A -85,B 0,C 180,E1 6995.066,E2 6995.066} C_VEL
LIN {X 0,Y 179.37,Z 528.567,A -85,B 0,C 180,E1 6992.408,E2 6992.408} C_VEL
LIN {X 0,Y 166.867,Z 542.359,A -85,B 0,C 180,E1 6988.96,E2 6988.96} C_VEL
LIN {X 0,Y 154.307,Z 554.44,A -85,B 0,C 180,E1 6984.725,E2 6984.725} C_VEL
LIN {X 0,Y 142.673,Z 564.372,A -85,B 0,C 180,E1 6979.803,E2 6979.803} C_VEL
LIN {X 0,Y 131.038,Z 573.268,A -85,B 0,C 180,E1 6973.368,E2 6973.368} C_VEL
LIN {X 0,Y 121.214,Z 580.155,A -85,B 0,C 180,E1 6965.845,E2 6965.845} C_VEL
LIN {X 0,Y 113.229,Z 585.445,A -85,B 0,C 180,E1 6956.762,E2 6956.762} C_VEL
LIN {X 0,Y 108.015,Z 588.886,A -85,B 0,C 180,E1 6946.672,E2 6946.672} C_VEL
LIN {X 0,Y 105.581,Z 590.599,A -85,B 0,C 180,E1 6935.976,E2 6935.976} C_VEL
LIN {X 0,Y 105.358,Z 590.744,A -85,B 0,C 180,E1 6926.732,E2 6926.732} C_VEL
LIN {X 0,Y 107.033,Z 589.538,A -85,B 0,C 180,E1 6916.299,E2 6916.299} C_VEL
LIN {X 0,Y 111.32,Z 586.697,A -85,B 0,C 180,E1 6906.157,E2 6906.157} C_VEL
LIN {X 0,Y 118.066,Z 582.297,A -85,B 0,C 180,E1 6897.177,E2 6897.177} C_VEL
LIN {X 0,Y 127.122,Z 576.145,A -85,B 0,C 180,E1 6889.242,E2 6889.242} C_VEL
LIN {X 0,Y 137.506,Z 568.556,A -85,B 0,C 180,E1 6882.739,E2 6882.739} C_VEL
LIN {X 0,Y 140.244,Z 566.293,A -85,B 0,C 180,E1 6881.164,E2 6881.164} C_VEL
LIN {X 0,Y 123.304,Z 568.939,A -85,B 0,C 180,E1 6871.809,E2 6871.809} C_VEL
LIN {X 0,Y 109.634,Z 571.462,A -85,B 0,C 180,E1 6855.88,E2 6855.88} C_VEL
LIN {X 0,Y 107.311,Z 572.283,A -85,B 0,C 180,E1 6849.927,E2 6849.927} C_VEL
LIN {X 0,Y 105.907,Z 573.203,A -85,B 0,C 180,E1 6844.333,E2 6844.333} C_VEL
LIN {X 0,Y 105.516,Z 574.752,A -85,B 0,C 180,E1 6835.926,E2 6835.926} C_VEL
LIN {X 0,Y 107.425,Z 582.159,A -85,B 0,C 180,E1 6826.546,E2 6826.546} C_VEL
LIN {X 0,Y 112.744,Z 589.127,A -85,B 0,C 180,E1 6815.925,E2 6815.925} C_VEL
LIN {X 0,Y 122.038,Z 594.567,A -85,B 0,C 180,E1 6806.144,E2 6806.144} C_VEL
LIN {X 0,Y 131.521,Z 597.636,A -85,B 0,C 180,E1 6799.746,E2 6799.746} C_VEL
LIN {X 0,Y 116.85,Z 597.99,A -85,B 0,C 180,E1 6788.66,E2 6788.66} C_VEL
LIN {X 0,Y 113.25,Z 597.926,A -85,B 0,C 180,E1 6784.409,E2 6784.409} C_VEL
LIN {X 0,Y 107.158,Z 603.05,A -85,B 0,C 180,E1 6774.243,E2 6774.243} C_VEL
LIN {X 0,Y 104.703,Z 606.208,A -85,B 0,C 180,E1 6763.816,E2 6763.816} C_VEL
LIN {X 0,Y 104.821,Z 607.659,A -85,B 0,C 180,E1 6754.38,E2 6754.38} C_VEL
LIN {X 0,Y 105.036,Z 607.833,A -85,B 0,C 180,E1 6748.913,E2 6748.913} C_VEL
LIN {X 0,Y 104.647,Z 607.399,A -85,B 0,C 180,E1 6743.079,E2 6743.079} C_VEL
LIN {X 0,Y 103.701,Z 606.771,A -85,B 0,C 180,E1 6739.169,E2 6739.169} C_VEL
LIN {X 0,Y 100.585,Z 605.153,A -85,B 0,C 180,E1 6732.538,E2 6732.538} C_VEL
LIN {X 0,Y 99.021,Z 603.223,A -85,B 0,C 180,E1 6726.234,E2 6726.234} C_VEL
LIN {X 0,Y 99.578,Z 602.179,A -85,B 0,C 180,E1 6723.409,E2 6723.409} C_VEL
LIN {X 0,Y 105.706,Z 597.103,A -85,B 0,C 180,E1 6712.749,E2 6712.749} C_VEL
LIN {X 0,Y 114.882,Z 590.16,A -85,B 0,C 180,E1 6703.436,E2 6703.436} C_VEL
LIN {X 0,Y 126.635,Z 581.129,A -85,B 0,C 180,E1 6695.591,E2 6695.591} C_VEL
LIN {X 0,Y 139.182,Z 570.823,A -85,B 0,C 180,E1 6689.635,E2 6689.635} C_VEL
LIN {X 0,Y 152.194,Z 559.024,A -85,B 0,C 180,E1 6684.965,E2 6684.965} C_VEL
LIN {X 0,Y 165.234,Z 545.745,A -85,B 0,C 180,E1 6681.277,E2 6681.277} C_VEL
LIN {X 0,Y 177.591,Z 531.462,A -85,B 0,C 180,E1 6678.444,E2 6678.444} C_VEL
LIN {X 0,Y 189.003,Z 516.334,A -85,B 0,C 180,E1 6676.234,E2 6676.234} C_VEL
LIN {X 0,Y 199.779,Z 499.767,A -85,B 0,C 180,E1 6674.443,E2 6674.443} C_VEL
LIN {X 0,Y 209.368,Z 482.349,A -85,B 0,C 180,E1 6673.047,E2 6673.047} C_VEL
LIN {X 0,Y 217.981,Z 463.409,A -85,B 0,C 180,E1 6671.931,E2 6671.931} C_VEL
LIN {X 0,Y 225.166,Z 443.506,A -85,B 0,C 180,E1 6671.09,E2 6671.09} C_VEL
LIN {X 0,Y 230.753,Z 422.689,A -85,B 0,C 180,E1 6670.464,E2 6670.464} C_VEL
LIN {X 0,Y 234.461,Z 401.647,A -85,B 0,C 180,E1 6669.98,E2 6669.98} C_VEL
LIN {X 0,Y 243.798,Z 318.45,A -85,B 0,C 180,E1 6668.371,E2 6668.371} C_VEL
LIN {X 0,Y 242.362,Z 314.385,A -85,B 0,C 180,E1 6665.682,E2 6665.682} C_VEL
LIN {X 0,Y 241.587,Z 312.285,A -85,B 0,C 180,E1 6663.796,E2 6663.796} C_VEL
LIN {X 0,Y 240.74,Z 309.636,A -85,B 0,C 180,E1 6660.475,E2 6660.475} C_VEL
LIN {X 0,Y 240.502,Z 309.386,A -85,B 0,C 180,E1 6655.708,E2 6655.708} C_VEL
LIN {X 0,Y 240.797,Z 310.08,A -85,B 0,C 180,E1 6653.682,E2 6653.682} C_VEL
LIN {X 0,Y 241.908,Z 313.634,A -85,B 0,C 180,E1 6649.882,E2 6649.882} C_VEL
LIN {X 0,Y 243.501,Z 318.437,A -85,B 0,C 180,E1 6646.645,E2 6646.645} C_VEL
LIN {X 0,Y 243.631,Z 319.195,A -85,B 0,C 180,E1 6646.371,E2 6646.371} C_VEL
LIN {X 0,Y 234.132,Z 404.244,A -85,B 0,C 180,E1 6644.817,E2 6644.817} C_VEL
LIN {X 0,Y 230.127,Z 424.449,A -85,B 0,C 180,E1 6644.255,E2 6644.255} C_VEL
LIN {X 0,Y 224.717,Z 443.459,A -85,B 0,C 180,E1 6643.499,E2 6643.499} C_VEL
LIN {X 0,Y 217.575,Z 462.492,A -85,B 0,C 180,E1 6642.463,E2 6642.463} C_VEL
LIN {X 0,Y 209.16,Z 480.362,A -85,B 0,C 180,E1 6641.169,E2 6641.169} C_VEL
LIN {X 0,Y 199.103,Z 497.921,A -85,B 0,C 180,E1 6639.477,E2 6639.477} C_VEL
LIN {X 0,Y 187.947,Z 514.214,A -85,B 0,C 180,E1 6637.363,E2 6637.363} C_VEL
LIN {X 0,Y 175.811,Z 529.274,A -85,B 0,C 180,E1 6634.717,E2 6634.717} C_VEL
LIN {X 0,Y 162.884,Z 543.04,A -85,B 0,C 180,E1 6631.373,E2 6631.373} C_VEL
LIN {X 0,Y 149.822,Z 555.109,A -85,B 0,C 180,E1 6627.228,E2 6627.228} C_VEL
LIN {X 0,Y 137.633,Z 565.034,A -85,B 0,C 180,E1 6622.354,E2 6622.354} C_VEL
LIN {X 0,Y 125.322,Z 573.923,A -85,B 0,C 180,E1 6615.889,E2 6615.889} C_VEL
LIN {X 0,Y 114.802,Z 580.808,A -85,B 0,C 180,E1 6608.193,E2 6608.193} C_VEL
LIN {X 0,Y 106.127,Z 586.096,A -85,B 0,C 180,E1 6598.713,E2 6598.713} C_VEL
LIN {X 0,Y 100.37,Z 589.535,A -85,B 0,C 180,E1 6587.984,E2 6587.984} C_VEL
LIN {X 0,Y 97.647,Z 591.246,A -85,B 0,C 180,E1 6576.463,E2 6576.463} C_VEL
LIN {X 0,Y 97.395,Z 591.39,A -85,B 0,C 180,E1 6566.465,E2 6566.465} C_VEL
LIN {X 0,Y 99.274,Z 590.188,A -85,B 0,C 180,E1 6555.218,E2 6555.218} C_VEL
LIN {X 0,Y 104.034,Z 587.346,A -85,B 0,C 180,E1 6544.371,E2 6544.371} C_VEL
LIN {X 0,Y 111.404,Z 582.949,A -85,B 0,C 180,E1 6534.938,E2 6534.938} C_VEL
LIN {X 0,Y 121.151,Z 576.799,A -85,B 0,C 180,E1 6526.761,E2 6526.761} C_VEL
LIN {X 0,Y 130.184,Z 570.568,A -85,B 0,C 180,E1 6521.136,E2 6521.136} C_VEL
LIN {X 0,Y 111.586,Z 573.329,A -85,B 0,C 180,E1 6508.939,E2 6508.939} C_VEL
LIN {X 0,Y 99.649,Z 576.104,A -85,B 0,C 180,E1 6489.239,E2 6489.239} C_VEL
LIN {X 0,Y 98.44,Z 577.02,A -85,B 0,C 180,E1 6482.912,E2 6482.912} C_VEL
LIN {X 0,Y 98.116,Z 578.319,A -85,B 0,C 180,E1 6475.325,E2 6475.325} C_VEL
LIN {X 0,Y 99.404,Z 580.112,A -85,B 0,C 180,E1 6466.625,E2 6466.625} C_VEL
LIN {X 0,Y 104.809,Z 587.686,A -85,B 0,C 180,E1 6455.182,E2 6455.182} C_VEL
LIN {X 0,Y 114.946,Z 593.976,A -85,B 0,C 180,E1 6444.353,E2 6444.353} C_VEL
LIN {X 0,Y 121.407,Z 596.447,A -85,B 0,C 180,E1 6439.627,E2 6439.627} C_VEL
LIN {X 0,Y 108.196,Z 596.156,A -85,B 0,C 180,E1 6428.597,E2 6428.597} C_VEL
LIN {X 0,Y 100.541,Z 601.707,A -85,B 0,C 180,E1 6417.87,E2 6417.87} C_VEL
LIN {X 0,Y 96.963,Z 605.286,A -85,B 0,C 180,E1 6406.17,E2 6406.17} C_VEL
LIN {X 0,Y 96.768,Z 606.975,A -85,B 0,C 180,E1 6395.34,E2 6395.34} C_VEL
LIN {X 0,Y 97.077,Z 607.214,A -85,B 0,C 180,E1 6389.414,E2 6389.414} C_VEL
LIN {X 0,Y 96.603,Z 606.632,A -85,B 0,C 180,E1 6381.672,E2 6381.672} C_VEL
LIN {X 0,Y 97.39,Z 604.572,A -85,B 0,C 180,E1 6370.821,E2 6370.821} C_VEL
LIN {X 0,Y 99.578,Z 602.179,A -85,B 0,C 180,E1 6363.409,E2 6363.409} C_VEL
LIN {X 0,Y 100.537,Z 600.483,A -85,B 0,C 180,E1 6359.108,E2 6359.108} C_VEL
LIN {X 0,Y 102.147,Z 594.929,A -85,B 0,C 180,E1 6347.508,E2 6347.508} C_VEL
LIN {X 0,Y 104.562,Z 592.757,A -85,B 0,C 180,E1 6344.278,E2 6344.278} C_VEL
LIN {X 0,Y 115.919,Z 584.854,A -85,B 0,C 180,E1 6335.832,E2 6335.832} C_VEL
LIN {X 0,Y 128.473,Z 575.549,A -85,B 0,C 180,E1 6329.355,E2 6329.355} C_VEL
LIN {X 0,Y 142.384,Z 564.149,A -85,B 0,C 180,E1 6324.098,E2 6324.098} C_VEL
LIN {X 0,Y 156.435,Z 551.138,A -85,B 0,C 180,E1 6320.031,E2 6320.031} C_VEL
LIN {X 0,Y 169.85,Z 536.966,A -85,B 0,C 180,E1 6316.953,E2 6316.953} C_VEL
LIN {X 0,Y 182.798,Z 521.154,A -85,B 0,C 180,E1 6314.511,E2 6314.511} C_VEL
LIN {X 0,Y 194.671,Z 504.18,A -85,B 0,C 180,E1 6312.623,E2 6312.623} C_VEL
LIN {X 0,Y 204.879,Z 486.892,A -85,B 0,C 180,E1 6311.219,E2 6311.219} C_VEL
LIN {X 0,Y 213.798,Z 468.685,A -85,B 0,C 180,E1 6310.133,E2 6310.133} C_VEL
LIN {X 0,Y 221.375,Z 449.517,A -85,B 0,C 180,E1 6309.305,E2 6309.305} C_VEL
LIN {X 0,Y 227.379,Z 429.711,A -85,B 0,C 180,E1 6308.691,E2 6308.691} C_VEL
LIN {X 0,Y 231.65,Z 409.655,A -85,B 0,C 180,E1 6308.216,E2 6308.216} C_VEL
LIN {X 0,Y 235.969,Z 375.21,A -85,B 0,C 180,E1 6307.571,E2 6307.571} C_VEL
LIN {X 0,Y 241.787,Z 323.973,A -85,B 0,C 180,E1 6306.649,E2 6306.649} C_VEL
LIN {X 0,Y 240.499,Z 320.169,A -85,B 0,C 180,E1 6303.575,E2 6303.575} C_VEL
LIN {X 0,Y 239.704,Z 317.531,A -85,B 0,C 180,E1 6300.239,E2 6300.239} C_VEL
LIN {X 0,Y 239.541,Z 317.371,A -85,B 0,C 180,E1 6295.451,E2 6295.451} C_VEL
LIN {X 0,Y 239.782,Z 318.102,A -85,B 0,C 180,E1 6293.775,E2 6293.775} C_VEL
LIN {X 0,Y 240.778,Z 321.473,A -85,B 0,C 180,E1 6290.197,E2 6290.197} C_VEL
LIN {X 0,Y 241.631,Z 324.642,A -85,B 0,C 180,E1 6288.142,E2 6288.142} C_VEL
LIN {X 0,Y 232.443,Z 404.698,A -85,B 0,C 180,E1 6286.735,E2 6286.735} C_VEL
LIN {X 0,Y 228.37,Z 424.814,A -85,B 0,C 180,E1 6286.204,E2 6286.204} C_VEL
LIN {X 0,Y 222.8,Z 443.992,A -85,B 0,C 180,E1 6285.483,E2 6285.483} C_VEL
LIN {X 0,Y 215.768,Z 462.396,A -85,B 0,C 180,E1 6284.542,E2 6284.542} C_VEL
LIN {X 0,Y 207.135,Z 480.448,A -85,B 0,C 180,E1 6283.316,E2 6283.316} C_VEL
LIN {X 0,Y 197.34,Z 497.287,A -85,B 0,C 180,E1 6281.799,E2 6281.799} C_VEL
LIN {X 0,Y 186.328,Z 513.188,A -85,B 0,C 180,E1 6279.889,E2 6279.889} C_VEL
LIN {X 0,Y 174.674,Z 527.529,A -85,B 0,C 180,E1 6277.579,E2 6277.579} C_VEL
LIN {X 0,Y 162.491,Z 540.476,A -85,B 0,C 180,E1 6274.755,E2 6274.755} C_VEL
LIN {X 0,Y 149.551,Z 552.43,A -85,B 0,C 180,E1 6271.138,E2 6271.138} C_VEL
LIN {X 0,Y 136.536,Z 562.929,A -85,B 0,C 180,E1 6266.592,E2 6266.592} C_VEL
LIN {X 0,Y 123.144,Z 572.393,A -85,B 0,C 180,E1 6260.47,E2 6260.47} C_VEL
LIN {X 0,Y 111.367,Z 579.779,A -85,B 0,C 180,E1 6253.021,E2 6253.021} C_VEL
LIN {X 0,Y 101.25,Z 585.551,A -85,B 0,C 180,E1 6243.569,E2 6243.569} C_VEL
LIN {X 0,Y 94.064,Z 589.438,A -85,B 0,C 180,E1 6232.494,E2 6232.494} C_VEL
LIN {X 0,Y 90.182,Z 591.577,A -85,B 0,C 180,E1 6220.214,E2 6220.214} C_VEL
LIN {X 0,Y 89.341,Z 592.118,A -85,B 0,C 180,E1 6208.713,E2 6208.713} C_VEL
LIN {X 0,Y 90.683,Z 591.358,A -85,B 0,C 180,E1 6197.256,E2 6197.256} C_VEL
LIN {X 0,Y 95.211,Z 588.904,A -85,B 0,C 180,E1 6185.157,E2 6185.157} C_VEL
LIN {X 0,Y 103.013,Z 584.679,A -85,B 0,C 180,E1 6174.378,E2 6174.378} C_VEL
LIN {X 0,Y 113.044,Z 578.892,A -85,B 0,C 180,E1 6165.669,E2 6165.669} C_VEL
LIN {X 0,Y 120.114,Z 574.535,A -85,B 0,C 180,E1 6161.12,E2 6161.12} C_VEL
LIN {X 0,Y 100.249,Z 577.425,A -85,B 0,C 180,E1 6145.397,E2 6145.397} C_VEL
LIN {X 0,Y 92.242,Z 579.513,A -85,B 0,C 180,E1 6129.359,E2 6129.359} C_VEL
LIN {X 0,Y 90.983,Z 580.453,A -85,B 0,C 180,E1 6122.521,E2 6122.521} C_VEL
LIN {X 0,Y 90.732,Z 581.637,A -85,B 0,C 180,E1 6114.944,E2 6114.944} C_VEL
LIN {X 0,Y 92.351,Z 583.618,A -85,B 0,C 180,E1 6104.297,E2 6104.297} C_VEL
LIN {X 0,Y 96.576,Z 585.596,A -85,B 0,C 180,E1 6094.884,E2 6094.884} C_VEL
LIN {X 0,Y 106.899,Z 592.59,A -85,B 0,C 180,E1 6083.231,E2 6083.231} C_VEL
LIN {X 0,Y 111.617,Z 594.628,A -85,B 0,C 180,E1 6079.595,E2 6079.595} C_VEL
LIN {X 0,Y 103.785,Z 594.342,A -85,B 0,C 180,E1 6073.162,E2 6073.162} C_VEL
LIN {X 0,Y 95.091,Z 599.909,A -85,B 0,C 180,E1 6063.15,E2 6063.15} C_VEL
LIN {X 0,Y 89.782,Z 603.996,A -85,B 0,C 180,E1 6050.7,E2 6050.7} C_VEL
LIN {X 0,Y 88.636,Z 606.157,A -85,B 0,C 180,E1 6037.784,E2 6037.784} C_VEL
LIN {X 0,Y 89.12,Z 606.589,A -85,B 0,C 180,E1 6030.004,E2 6030.004} C_VEL
LIN {X 0,Y 88.638,Z 606.142,A -85,B 0,C 180,E1 6022.225,E2 6022.225} C_VEL
LIN {X 0,Y 89.424,Z 604.194,A -85,B 0,C 180,E1 6010.406,E2 6010.406} C_VEL
LIN {X 0,Y 93.564,Z 600.498,A -85,B 0,C 180,E1 5998.429,E2 5998.429} C_VEL
LIN {X 0,Y 101.093,Z 595.117,A -85,B 0,C 180,E1 5987.741,E2 5987.741} C_VEL
LIN {X 0,Y 104.562,Z 592.757,A -85,B 0,C 180,E1 5984.278,E2 5984.278} C_VEL
LIN {X 0,Y 107.627,Z 590.132,A -85,B 0,C 180,E1 5980.7,E2 5980.7} C_VEL
LIN {X 0,Y 114.098,Z 582.807,A -85,B 0,C 180,E1 5971.575,E2 5971.575} C_VEL
LIN {X 0,Y 118.244,Z 579.414,A -85,B 0,C 180,E1 5968.801,E2 5968.801} C_VEL
LIN {X 0,Y 131.792,Z 569.438,A -85,B 0,C 180,E1 5963.375,E2 5963.375} C_VEL
LIN {X 0,Y 145.998,Z 557.627,A -85,B 0,C 180,E1 5959.085,E2 5959.085} C_VEL
LIN {X 0,Y 160.003,Z 544.32,A -85,B 0,C 180,E1 5955.782,E2 5955.782} C_VEL
LIN {X 0,Y 173.559,Z 529.467,A -85,B 0,C 180,E1 5953.207,E2 5953.207} C_VEL
LIN {X 0,Y 186.029,Z 513.543,A -85,B 0,C 180,E1 5951.231,E2 5951.231} C_VEL
LIN {X 0,Y 197.065,Z 496.973,A -85,B 0,C 180,E1 5949.738,E2 5949.738} C_VEL
LIN {X 0,Y 206.734,Z 479.711,A -85,B 0,C 180,E1 5948.594,E2 5948.594} C_VEL
LIN {X 0,Y 214.915,Z 462.058,A -85,B 0,C 180,E1 5947.731,E2 5947.731} C_VEL
LIN {X 0,Y 222.137,Z 442.536,A -85,B 0,C 180,E1 5947.042,E2 5947.042} C_VEL
LIN {X 0,Y 227.808,Z 421.914,A -85,B 0,C 180,E1 5946.518,E2 5946.518} C_VEL
LIN {X 0,Y 231.597,Z 401.018,A -85,B 0,C 180,E1 5946.095,E2 5946.095} C_VEL
LIN {X 0,Y 239.933,Z 329.823,A -85,B 0,C 180,E1 5944.846,E2 5944.846} C_VEL
LIN {X 0,Y 239.199,Z 327.479,A -85,B 0,C 180,E1 5942.635,E2 5942.635} C_VEL
LIN {X 0,Y 238.684,Z 325.429,A -85,B 0,C 180,E1 5940,E2 5940} C_VEL
LIN {X 0,Y 238.597,Z 325.367,A -85,B 0,C 180,E1 5935.192,E2 5935.192} C_VEL
LIN {X 0,Y 238.809,Z 326.335,A -85,B 0,C 180,E1 5933.629,E2 5933.629} C_VEL
LIN {X 0,Y 239.662,Z 329.312,A -85,B 0,C 180,E1 5930.514,E2 5930.514} C_VEL
LIN {X 0,Y 239.843,Z 330.296,A -85,B 0,C 180,E1 5929.936,E2 5929.936} C_VEL
LIN {X 0,Y 231.048,Z 404.99,A -85,B 0,C 180,E1 5928.681,E2 5928.681} C_VEL
LIN {X 0,Y 226.894,Z 425.135,A -85,B 0,C 180,E1 5928.183,E2 5928.183} C_VEL
LIN {X 0,Y 221.2,Z 444.389,A -85,B 0,C 180,E1 5927.506,E2 5927.506} C_VEL
LIN {X 0,Y 213.789,Z 463.383,A -85,B 0,C 180,E1 5926.593,E2 5926.593} C_VEL
LIN {X 0,Y 204.58,Z 482.084,A -85,B 0,C 180,E1 5925.389,E2 5925.389} C_VEL
LIN {X 0,Y 194.092,Z 499.488,A -85,B 0,C 180,E1 5923.886,E2 5923.886} C_VEL
LIN {X 0,Y 182.848,Z 515.129,A -85,B 0,C 180,E1 5922.071,E2 5922.071} C_VEL
LIN {X 0,Y 170.144,Z 530.11,A -85,B 0,C 180,E1 5919.713,E2 5919.713} C_VEL
LIN {X 0,Y 156.697,Z 543.643,A -85,B 0,C 180,E1 5916.75,E2 5916.75} C_VEL
LIN {X 0,Y 142.598,Z 555.824,A -85,B 0,C 180,E1 5912.929,E2 5912.929} C_VEL
LIN {X 0,Y 128.462,Z 566.355,A -85,B 0,C 180,E1 5908.03,E2 5908.03} C_VEL
LIN {X 0,Y 114.726,Z 575.23,A -85,B 0,C 180,E1 5901.657,E2 5901.657} C_VEL
LIN {X 0,Y 102.659,Z 582.113,A -85,B 0,C 180,E1 5893.745,E2 5893.745} C_VEL
LIN {X 0,Y 92.374,Z 587.396,A -85,B 0,C 180,E1 5883.501,E2 5883.501} C_VEL
LIN {X 0,Y 85.281,Z 590.832,A -85,B 0,C 180,E1 5871.308,E2 5871.308} C_VEL
LIN {X 0,Y 81.803,Z 592.538,A -85,B 0,C 180,E1 5857.722,E2 5857.722} C_VEL
LIN {X 0,Y 81.476,Z 592.68,A -85,B 0,C 180,E1 5845.773,E2 5845.773} C_VEL
LIN {X 0,Y 83.887,Z 591.488,A -85,B 0,C 180,E1 5832.47,E2 5832.47} C_VEL
LIN {X 0,Y 89.837,Z 588.643,A -85,B 0,C 180,E1 5819.94,E2 5819.94} C_VEL
LIN {X 0,Y 98.689,Z 584.25,A -85,B 0,C 180,E1 5809.574,E2 5809.574} C_VEL
LIN {X 0,Y 109.969,Z 578.099,A -85,B 0,C 180,E1 5800.971,E2 5800.971} C_VEL
LIN {X 0,Y 93.197,Z 580.484,A -85,B 0,C 180,E1 5786.783,E2 5786.783} C_VEL
LIN {X 0,Y 84.736,Z 582.612,A -85,B 0,C 180,E1 5769.51,E2 5769.51} C_VEL
LIN {X 0,Y 83.542,Z 583.477,A -85,B 0,C 180,E1 5762.745,E2 5762.745} C_VEL
LIN {X 0,Y 83.289,Z 584.557,A -85,B 0,C 180,E1 5755.181,E2 5755.181} C_VEL
LIN {X 0,Y 85.118,Z 586.627,A -85,B 0,C 180,E1 5742.924,E2 5742.924} C_VEL
LIN {X 0,Y 98.938,Z 590.808,A -85,B 0,C 180,E1 5721.943,E2 5721.943} C_VEL
LIN {X 0,Y 101.804,Z 592.254,A -85,B 0,C 180,E1 5719.374,E2 5719.374} C_VEL
LIN {X 0,Y 100.435,Z 592.294,A -85,B 0,C 180,E1 5718.306,E2 5718.306} C_VEL
LIN {X 0,Y 90.095,Z 598.18,A -85,B 0,C 180,E1 5708.429,E2 5708.429} C_VEL
LIN {X 0,Y 83.11,Z 602.58,A -85,B 0,C 180,E1 5695.669,E2 5695.669} C_VEL
LIN {X 0,Y 80.615,Z 605.168,A -85,B 0,C 180,E1 5681.451,E2 5681.451} C_VEL
LIN {X 0,Y 81.073,Z 605.899,A -85,B 0,C 180,E1 5671.418,E2 5671.418} C_VEL
LIN {X 0,Y 80.822,Z 605.736,A -85,B 0,C 180,E1 5665.037,E2 5665.037} C_VEL
LIN {X 0,Y 81.111,Z 604.198,A -85,B 0,C 180,E1 5652.055,E2 5652.055} C_VEL
LIN {X 0,Y 84.991,Z 600.977,A -85,B 0,C 180,E1 5638.832,E2 5638.832} C_VEL
LIN {X 0,Y 93.08,Z 595.756,A -85,B 0,C 180,E1 5626.575,E2 5626.575} C_VEL
LIN {X 0,Y 103.913,Z 588.991,A -85,B 0,C 180,E1 5617.006,E2 5617.006} C_VEL
LIN {X 0,Y 117.029,Z 580.292,A -85,B 0,C 180,E1 5609.379,E2 5609.379} C_VEL
LIN {X 0,Y 118.244,Z 579.414,A -85,B 0,C 180,E1 5608.801,E2 5608.801} C_VEL
LIN {X 0,Y 122.604,Z 575.909,A -85,B 0,C 180,E1 5606.247,E2 5606.247} C_VEL
LIN {X 0,Y 132.203,Z 566.532,A -85,B 0,C 180,E1 5599.478,E2 5599.478} C_VEL
LIN {X 0,Y 137.009,Z 562.305,A -85,B 0,C 180,E1 5597.613,E2 5597.613} C_VEL
LIN {X 0,Y 151.584,Z 549.706,A -85,B 0,C 180,E1 5594.171,E2 5594.171} C_VEL
LIN {X 0,Y 165.345,Z 536.003,A -85,B 0,C 180,E1 5591.598,E2 5591.598} C_VEL
LIN {X 0,Y 178.927,Z 520.222,A -85,B 0,C 180,E1 5589.51,E2 5589.51} C_VEL
LIN {X 0,Y 190.811,Z 503.981,A -85,B 0,C 180,E1 5587.975,E2 5587.975} C_VEL
LIN {X 0,Y 201.861,Z 485.992,A -85,B 0,C 180,E1 5586.745,E2 5586.745} C_VEL
LIN {X 0,Y 211.361,Z 467.149,A -85,B 0,C 180,E1 5585.82,E2 5585.82} C_VEL
LIN {X 0,Y 219.095,Z 447.932,A -85,B 0,C 180,E1 5585.148,E2 5585.148} C_VEL
LIN {X 0,Y 225.353,Z 427.46,A -85,B 0,C 180,E1 5584.634,E2 5584.634} C_VEL
LIN {X 0,Y 229.782,Z 406.314,A -85,B 0,C 180,E1 5584.217,E2 5584.217} C_VEL
LIN {X 0,Y 238.322,Z 335.872,A -85,B 0,C 180,E1 5583.041,E2 5583.041} C_VEL
LIN {X 0,Y 237.67,Z 333.328,A -85,B 0,C 180,E1 5579.758,E2 5579.758} C_VEL
LIN {X 0,Y 237.624,Z 333.319,A -85,B 0,C 180,E1 5575.172,E2 5575.172} C_VEL
LIN {X 0,Y 238.24,Z 336.214,A -85,B 0,C 180,E1 5571.751,E2 5571.751} C_VEL
LIN {X 0,Y 229.892,Z 405.443,A -85,B 0,C 180,E1 5570.646,E2 5570.646} C_VEL
LIN {X 0,Y 225.642,Z 425.64,A -85,B 0,C 180,E1 5570.18,E2 5570.18} C_VEL
LIN {X 0,Y 219.857,Z 444.853,A -85,B 0,C 180,E1 5569.553,E2 5569.553} C_VEL
LIN {X 0,Y 212.372,Z 463.719,A -85,B 0,C 180,E1 5568.714,E2 5568.714} C_VEL
LIN {X 0,Y 203.187,Z 482.115,A -85,B 0,C 180,E1 5567.622,E2 5567.622} C_VEL
LIN {X 0,Y 192.497,Z 499.603,A -85,B 0,C 180,E1 5566.232,E2 5566.232} C_VEL
LIN {X 0,Y 180.551,Z 515.869,A -85,B 0,C 180,E1 5564.48,E2 5564.48} C_VEL
LIN {X 0,Y 167.581,Z 530.775,A -85,B 0,C 180,E1 5562.284,E2 5562.284} C_VEL
LIN {X 0,Y 153.715,Z 544.329,A -85,B 0,C 180,E1 5559.492,E2 5559.492} C_VEL
LIN {X 0,Y 139.134,Z 556.493,A -85,B 0,C 180,E1 5555.868,E2 5555.868} C_VEL
LIN {X 0,Y 124.401,Z 567.015,A -85,B 0,C 180,E1 5551.166,E2 5551.166} C_VEL
LIN {X 0,Y 109.926,Z 575.884,A -85,B 0,C 180,E1 5544.94,E2 5544.94} C_VEL
LIN {X 0,Y 97.017,Z 582.764,A -85,B 0,C 180,E1 5537.026,E2 5537.026} C_VEL
LIN {X 0,Y 85.795,Z 588.046,A -85,B 0,C 180,E1 5526.461,E2 5526.461} C_VEL
LIN {X 0,Y 77.874,Z 591.481,A -85,B 0,C 180,E1 5513.449,E2 5513.449} C_VEL
LIN {X 0,Y 73.901,Z 593.184,A -85,B 0,C 180,E1 5498.554,E2 5498.554} C_VEL
LIN {X 0,Y 73.522,Z 593.325,A -85,B 0,C 180,E1 5485.315,E2 5485.315} C_VEL
LIN {X 0,Y 76.28,Z 592.141,A -85,B 0,C 180,E1 5470.698,E2 5470.698} C_VEL
LIN {X 0,Y 82.992,Z 589.293,A -85,B 0,C 180,E1 5457.165,E2 5457.165} C_VEL
LIN {X 0,Y 93.126,Z 584.701,A -85,B 0,C 180,E1 5446.003,E2 5446.003} C_VEL
LIN {X 0,Y 99.659,Z 581.441,A -85,B 0,C 180,E1 5440.875,E2 5440.875} C_VEL
LIN {X 0,Y 77.328,Z 585.352,A -85,B 0,C 180,E1 5410.431,E2 5410.431} C_VEL
LIN {X 0,Y 76.003,Z 586.219,A -85,B 0,C 180,E1 5403.018,E2 5403.018} C_VEL
LIN {X 0,Y 75.705,Z 587.295,A -85,B 0,C 180,E1 5394.697,E2 5394.697} C_VEL
LIN {X 0,Y 77.657,Z 589.213,A -85,B 0,C 180,E1 5382.002,E2 5382.002} C_VEL
LIN {X 0,Y 92.062,Z 593.254,A -85,B 0,C 180,E1 5359.732,E2 5359.732} C_VEL
LIN {X 0,Y 81.421,Z 598.814,A -85,B 0,C 180,E1 5348.782,E2 5348.782} C_VEL
LIN {X 0,Y 74.556,Z 602.778,A -85,B 0,C 180,E1 5334.571,E2 5334.571} C_VEL
LIN {X 0,Y 72.639,Z 604.929,A -85,B 0,C 180,E1 5318.714,E2 5318.714} C_VEL
LIN {X 0,Y 73.163,Z 605.298,A -85,B 0,C 180,E1 5310.005,E2 5310.005} C_VEL
LIN {X 0,Y 72.62,Z 604.747,A -85,B 0,C 180,E1 5299.694,E2 5299.694} C_VEL
LIN {X 0,Y 74.603,Z 602.579,A -85,B 0,C 180,E1 5284.609,E2 5284.609} C_VEL
LIN {X 0,Y 81.26,Z 598.473,A -85,B 0,C 180,E1 5270.227,E2 5270.227} C_VEL
LIN {X 0,Y 92.45,Z 592.185,A -85,B 0,C 180,E1 5258.057,E2 5258.057} C_VEL
LIN {X 0,Y 105.582,Z 584.441,A -85,B 0,C 180,E1 5249.405,E2 5249.405} C_VEL
LIN {X 0,Y 120.403,Z 574.752,A -85,B 0,C 180,E1 5242.822,E2 5242.822} C_VEL
LIN {X 0,Y 135.607,Z 563.456,A -85,B 0,C 180,E1 5237.993,E2 5237.993} C_VEL
LIN {X 0,Y 137.009,Z 562.305,A -85,B 0,C 180,E1 5237.613,E2 5237.613} C_VEL
LIN {X 0,Y 141.882,Z 557.965,A -85,B 0,C 180,E1 5235.897,E2 5235.897} C_VEL
LIN {X 0,Y 152.769,Z 546.602,A -85,B 0,C 180,E1 5230.998,E2 5230.998} C_VEL
LIN {X 0,Y 157.632,Z 541.588,A -85,B 0,C 180,E1 5229.759,E2 5229.759} C_VEL
LIN {X 0,Y 171.533,Z 526.85,A -85,B 0,C 180,E1 5227.704,E2 5227.704} C_VEL
LIN {X 0,Y 184.031,Z 511.349,A -85,B 0,C 180,E1 5226.166,E2 5226.166} C_VEL
LIN {X 0,Y 195.693,Z 494.198,A -85,B 0,C 180,E1 5224.945,E2 5224.945} C_VEL
LIN {X 0,Y 205.968,Z 475.968,A -85,B 0,C 180,E1 5224.011,E2 5224.011} C_VEL
LIN {X 0,Y 214.644,Z 456.971,A -85,B 0,C 180,E1 5223.315,E2 5223.315} C_VEL
LIN {X 0,Y 221.727,Z 437.083,A -85,B 0,C 180,E1 5222.805,E2 5222.805} C_VEL
LIN {X 0,Y 227.094,Z 416.292,A -85,B 0,C 180,E1 5222.398,E2 5222.398} C_VEL
LIN {X 0,Y 230.573,Z 394.956,A -85,B 0,C 180,E1 5222.046,E2 5222.046} C_VEL
LIN {X 0,Y 236.879,Z 342.467,A -85,B 0,C 180,E1 5221.209,E2 5221.209} C_VEL
LIN {X 0,Y 236.659,Z 341.229,A -85,B 0,C 180,E1 5219.515,E2 5219.515} C_VEL
LIN {X 0,Y 236.664,Z 341.321,A -85,B 0,C 180,E1 5215.031,E2 5215.031} C_VEL
LIN {X 0,Y 236.809,Z 342.717,A -85,B 0,C 180,E1 5213.581,E2 5213.581} C_VEL
LIN {X 0,Y 229.039,Z 405.731,A -85,B 0,C 180,E1 5212.632,E2 5212.632} C_VEL
LIN {X 0,Y 224.735,Z 425.897,A -85,B 0,C 180,E1 5212.203,E2 5212.203} C_VEL
LIN {X 0,Y 218.797,Z 445.315,A -85,B 0,C 180,E1 5211.622,E2 5211.622} C_VEL
LIN {X 0,Y 211.15,Z 464.273,A -85,B 0,C 180,E1 5210.849,E2 5210.849} C_VEL
LIN {X 0,Y 202.107,Z 482.128,A -85,B 0,C 180,E1 5209.883,E2 5209.883} C_VEL
LIN {X 0,Y 191.229,Z 499.705,A -85,B 0,C 180,E1 5208.614,E2 5208.614} C_VEL
LIN {X 0,Y 179.048,Z 516.044,A -85,B 0,C 180,E1 5207.013,E2 5207.013} C_VEL
LIN {X 0,Y 165.634,Z 531.167,A -85,B 0,C 180,E1 5204.973,E2 5204.973} C_VEL
LIN {X 0,Y 151.098,Z 545.012,A -85,B 0,C 180,E1 5202.334,E2 5202.334} C_VEL
LIN {X 0,Y 136.055,Z 557.161,A -85,B 0,C 180,E1 5198.949,E2 5198.949} C_VEL
LIN {X 0,Y 120.634,Z 567.735,A -85,B 0,C 180,E1 5194.468,E2 5194.468} C_VEL
LIN {X 0,Y 105.519,Z 576.538,A -85,B 0,C 180,E1 5188.511,E2 5188.511} C_VEL
LIN {X 0,Y 91.731,Z 583.416,A -85,B 0,C 180,E1 5180.698,E2 5180.698} C_VEL
LIN {X 0,Y 79.412,Z 588.722,A -85,B 0,C 180,E1 5169.82,E2 5169.82} C_VEL
LIN {X 0,Y 70.597,Z 592.129,A -85,B 0,C 180,E1 5156.037,E2 5156.037} C_VEL
LIN {X 0,Y 66.018,Z 593.831,A -85,B 0,C 180,E1 5139.584,E2 5139.584} C_VEL
LIN {X 0,Y 65.52,Z 593.991,A -85,B 0,C 180,E1 5125.618,E2 5125.618} C_VEL
LIN {X 0,Y 68.45,Z 592.916,A -85,B 0,C 180,E1 5109.472,E2 5109.472} C_VEL
LIN {X 0,Y 75.426,Z 590.332,A -85,B 0,C 180,E1 5095.243,E2 5095.243} C_VEL
LIN {X 0,Y 86.458,Z 585.842,A -85,B 0,C 180,E1 5083.227,E2 5083.227} C_VEL
LIN {X 0,Y 89.394,Z 584.472,A -85,B 0,C 180,E1 5080.685,E2 5080.685} C_VEL
LIN {X 0,Y 69.669,Z 587.937,A -85,B 0,C 180,E1 5050.754,E2 5050.754} C_VEL
LIN {X 0,Y 68.14,Z 589.483,A -85,B 0,C 180,E1 5036.28,E2 5036.28} C_VEL
LIN {X 0,Y 70.593,Z 591.762,A -85,B 0,C 180,E1 5019.21,E2 5019.21} C_VEL
LIN {X 0,Y 82.198,Z 594.927,A -85,B 0,C 180,E1 5000.032,E2 5000.032} C_VEL
LIN {X 0,Y 71.413,Z 599.964,A -85,B 0,C 180,E1 4987.023,E2 4987.023} C_VEL
LIN {X 0,Y 65.503,Z 603.175,A -85,B 0,C 180,E1 4970.559,E2 4970.559} C_VEL
LIN {X 0,Y 64.881,Z 604.507,A -85,B 0,C 180,E1 4954.425,E2 4954.425} C_VEL
LIN {X 0,Y 65.078,Z 604.599,A -85,B 0,C 180,E1 4948.245,E2 4948.245} C_VEL
LIN {X 0,Y 64.799,Z 603.749,A -85,B 0,C 180,E1 4934.799,E2 4934.799} C_VEL
LIN {X 0,Y 68.773,Z 601.008,A -85,B 0,C 180,E1 4917.464,E2 4917.464} C_VEL
LIN {X 0,Y 77.754,Z 596.429,A -85,B 0,C 180,E1 4902.871,E2 4902.871} C_VEL
LIN {X 0,Y 90.503,Z 589.929,A -85,B 0,C 180,E1 4891.723,E2 4891.723} C_VEL
LIN {X 0,Y 104.956,Z 581.843,A -85,B 0,C 180,E1 4883.869,E2 4883.869} C_VEL
LIN {X 0,Y 120.028,Z 572.286,A -85,B 0,C 180,E1 4878.271,E2 4878.271} C_VEL
LIN {X 0,Y 135.442,Z 561.041,A -85,B 0,C 180,E1 4874.099,E2 4874.099} C_VEL
LIN {X 0,Y 149.783,Z 548.99,A -85,B 0,C 180,E1 4871.117,E2 4871.117} C_VEL
LIN {X 0,Y 157.632,Z 541.588,A -85,B 0,C 180,E1 4869.759,E2 4869.759} C_VEL
LIN {X 0,Y 162.473,Z 536.483,A -85,B 0,C 180,E1 4868.616,E2 4868.616} C_VEL
LIN {X 0,Y 173.379,Z 523.198,A -85,B 0,C 180,E1 4865.015,E2 4865.015} C_VEL
LIN {X 0,Y 177.913,Z 517.465,A -85,B 0,C 180,E1 4864.176,E2 4864.176} C_VEL
LIN {X 0,Y 189.887,Z 501.379,A -85,B 0,C 180,E1 4863.018,E2 4863.018} C_VEL
LIN {X 0,Y 200.602,Z 484.212,A -85,B 0,C 180,E1 4862.126,E2 4862.126} C_VEL
LIN {X 0,Y 210.029,Z 465.83,A -85,B 0,C 180,E1 4861.439,E2 4861.439} C_VEL
LIN {X 0,Y 217.99,Z 446.307,A -85,B 0,C 180,E1 4860.925,E2 4860.925} C_VEL
LIN {X 0,Y 224.252,Z 425.907,A -85,B 0,C 180,E1 4860.538,E2 4860.538} C_VEL
LIN {X 0,Y 228.625,Z 405.131,A -85,B 0,C 180,E1 4860.207,E2 4860.207} C_VEL
LIN {X 0,Y 235.665,Z 349.149,A -85,B 0,C 180,E1 4859.37,E2 4859.37} C_VEL
LIN {X 0,Y 235.628,Z 349.272,A -85,B 0,C 180,E1 4855.43,E2 4855.43} C_VEL
LIN {X 0,Y 228.432,Z 406.184,A -85,B 0,C 180,E1 4854.627,E2 4854.627} C_VEL
LIN {X 0,Y 224.05,Z 426.368,A -85,B 0,C 180,E1 4854.235,E2 4854.235} C_VEL
LIN {X 0,Y 218.001,Z 445.84,A -85,B 0,C 180,E1 4853.706,E2 4853.706} C_VEL
LIN {X 0,Y 210.517,Z 464.187,A -85,B 0,C 180,E1 4853.033,E2 4853.033} C_VEL
LIN {X 0,Y 200.862,Z 482.997,A -85,B 0,C 180,E1 4852.117,E2 4852.117} C_VEL
